// TwinCAT 3 PLC project FLC
// ProgramVersion: 3.1.4026.12
// CompilerDefines: ABG
// libraries:
//   Tc2_IoFunctions, * (Beckhoff Automation GmbH)
//   Tc2_ModbusSrv, * (Beckhoff Automation GmbH)
//   Tc2_Standard, * (Beckhoff Automation GmbH)
//   Tc2_System, * (Beckhoff Automation GmbH)
//   Tc2_Utilities, * (Beckhoff Automation GmbH)
//   Tc3_Module, * (Beckhoff Automation GmbH)
//   EAP_Controller,1.0,LUA
//   Modbus_SPC,1.0,LUA
// project tree:
//   Functions/Communications/ EtherCAT_MappingEAP.TcPOU, EtherCAT_MappingModbus.TcPOU, Mapping_Monitoring_Variables.TcPOU, Mapping_Monitoring_Variables_ABG.TcPOU, Remap_EtherCAT_Variables.TcPOU
//   Functions/EventRecoder/ HistorianFunctionBlock.TcPOU, UnixTimestamp.TcPOU
//   Functions/Filters/ BandPassFilter.TcPOU, BandPassFilterParameters.TcPOU, BandPassFilterStruct.TcDUT, HighPassFilter.TcDUT, HPF_FilterInit.TcPOU, HPF_Function.TcPOU, LowPassFilter.TcDUT, LPF_FilterInit.TcPOU, LPF_Function.TcPOU
//   Functions/ Mapping_ModbusReadRegisters.TcPOU, Mapping_ModbusWriteRegisters.TcPOU, ModReadScaling.TcPOU
//   GlobalVar/ Communications.TcGVL, GlobalVar.TcGVL, GVL.TcGVL
//   Programs/ EAPControl.TcPOU, Timer.TcPOU, ModbusControl_Comm.TcPOU, State_Machine.TcPOU
//   Structures/Communication/EtherCAT/EAP Based Controller/EtherCAT/Commands Per Service/ AdditionalService_Struct_EAP.TcDUT, CommonBlock_Struct_EAP.TcDUT, FreqRegulation_Struct_EAP.TcDUT, InertiaEmulation_Struct_EAP.TcDUT, ModalFreq_Struct_EAP.TcDUT, VoltageRegulation_Struct_EAP.TcDUT
//   Structures/Communication/EtherCAT/EAP Based Controller/EtherCAT/Commands Per Service/Bits Per Commands/ Bits_AdditionalService_EAP.TcDUT, Bits_CommonBlock_EAP.TcDUT, Bits_FreqRegulation_EAP.TcDUT, Bits_InertiaEmulation_EAP.TcDUT, Bits_ModalFreq_EAP.TcDUT, Bits_VoltageRegulation_EAP.TcDUT
//   Structures/Communication/EtherCAT/EAP Based Controller/EtherCAT/ Commands_EAP.TcDUT, Parameters_EAP.TcDUT
//   Structures/Communication/EtherCAT/EAP Based Controller/EtherCAT/Parameters Per Service/ AdditionalService_Param_Struct_EAP.TcDUT, CommonBlock_Param_Struct_EAP.TcDUT, FreqRegulation_Param_Struct_EAP.TcDUT, InertiaEmulation_Param_Struct_EAP.TcDUT, ModalFreq_Param_Struct_EAP.TcDUT, VoltageRegulation_Param_Struct_EAP.TcDUT
//   Structures/Communication/EtherCAT/ EtherCAT_Inputs.TcDUT, EtherCAT_Monitor_Variables.TcDUT, EtherCAT_Stat_Variables.TcDUT, PowerOfService_Struct.TcDUT
//   Structures/Communication/EtherCAT/Modbus Based Controller/EtherCAT/Commands Per Service/ AdditionalService_Struct.TcDUT, CommonBlock_Struct.TcDUT, FreqRegulation_Struct.TcDUT, InertiaEmulation_Struct.TcDUT, ModalFreq_Struct.TcDUT, VoltageRegulation_Struct.TcDUT
//   Structures/Communication/EtherCAT/Modbus Based Controller/EtherCAT/Commands Per Service/Bits Per Commands/ Bits_AdditionalService.TcDUT, Bits_CommonBlock.TcDUT, Bits_FreqRegulation.TcDUT, Bits_InertiaEmulation.TcDUT, Bits_ModalFreq.TcDUT, Bits_VoltageRegulation.TcDUT
//   Structures/Communication/EtherCAT/Modbus Based Controller/EtherCAT/ Commands.TcDUT, Parameters.TcDUT
//   Structures/Communication/EtherCAT/Modbus Based Controller/EtherCAT/Parameters Per Service/ AdditionalService_Param_Struct.TcDUT, CommonBlock_Param_Struct.TcDUT, FreqRegulation_Param_Struct.TcDUT, InertiaEmulation_Param_Struct.TcDUT, ModalFreq_Param_Struct.TcDUT, VoltageRegulation_Param_Struct.TcDUT
//   Structures/Communication/EtherCAT/Modbus Based Controller/ EtherCAT_INT_VALUES.TcDUT
//   Structures/Communication/EtherCAT/RemapForSLC/EAP_para/ AdditionalService_Param_Struct_EAP_DINT.TcDUT, CommonBlock_Param_Struct_EAP_DINT.TcDUT, FreqRegulation_Param_Struct_EAP_DINT.TcDUT, InertiaEmulation_Param_Struct_EAP_DINT.TcDUT, ModalFreq_Param_Struct_EAP_DINT.TcDUT, VoltageRegulation_Param_Struct_EAP_DINT.TcDUT
//   Structures/Communication/EtherCAT/RemapForSLC/ EtherCAT_Inputs_DINT.TcDUT, EtherCAT_Monitor_Variables_DINT.TcDUT, Parameters_DINT.TcDUT, Parameters_EAP_DINT.TcDUT
//   Structures/Communication/EtherCAT/RemapForSLC/Modbus_para/ AdditionalService_Param_Struct_DINT.TcDUT, CommonBlock_Param_Struct_DINT.TcDUT, FreqRegulation_Param_Struct_DINT.TcDUT, InertiaEmulation_Param_Struct_DINT.TcDUT, ModalFreq_Param_Struct_DINT.TcDUT, VoltageRegulation_Param_Struct_DINT.TcDUT
//   Structures/Communication/EtherCAT/Warning/ Warnings_FLC.TcDUT, Warning_FLC_DINT.TcDUT
//   Structures/Communication/Modbus/ ModbusHoldingRegs.TcDUT, ModbusRead.TcDUT, ModbusRead_NRG.TcDUT, ModbusWrite.TcDUT, ModbusWrite_NRG.TcDUT, ScaledModRead.TcDUT
//   Structures/EventRecorder/ EthercatDataPacket.TcDUT
//   Structures/EventRecorder/HistorianDataType/ DateTimetype.TcDUT
//   Structures/StateMachine/ eCurrentState.TcDUT, eFEC_CurrState.TcDUT, StateMachineCommand.TcDUT
//   Structures/Transformations/ abcSignal.TcDUT, alphabetaSignal.TcDUT, dqsignal.TcDUT
//   Tasks/ EAPControl_Task.TcTTO, ModbusComm.TcTTO, StateMachine.TcTTO, TimerTask.TcTTO
// real-time tasks:
//   TASK StateMachine: cycle T#5ms, priority 8, ADS port 350
//   TASK ModbusComm: cycle T#20ms, priority 12, ADS port 351
//   TASK TimerTask: cycle T#1ms, priority 6, ADS port 353
//   TASK EAPControl_Task: cycle T#800us, priority 4, ADS port 354
//   TASK PlcTask: cycle T#10ms, priority 10, ADS port 352
// I/O:
//   DEVICE Device 1 (EtherCAT Slave), AmsNetId 10.150.0.126.2.255
// variable links:
//   FLC/FLC Instance <-> Device 1 (EtherCAT Slave)
//     EAPControl_Task Inputs/Communications.EtherCAT_Commands <-> Inputs/Commands Modbus
//     ModbusComm Inputs/Communications.EtherCAT_EAP_Commands <-> Inputs/Commands EAP
//     StateMachine Inputs/Communications.EhterCAT_Parameters_DINT <-> Inputs/Modbus_parameters
//     StateMachine Inputs/Communications.EtherCAT_EAP_Parameters_DINT <-> Inputs/EAP_paramteres
//     StateMachine Inputs/Communications.EtherCAT_Inputs_DINT <-> Inputs/EtherCAT_inputs
//     StateMachine Outputs/Communications.EtherCAT_Monitor_Variables_DINT <-> Outputs/Mornitoring Information
//     StateMachine Outputs/Communications.EtherCAT_Variables <-> Outputs/Status
//     StateMachine Outputs/Communications.PowerOfService <-> Outputs/PowerOfservices
//     TimerTask Inputs/GVL.TransmitApproved <-> Inputs/EventRecorderApproved
//     TimerTask Outputs/GVL.HistorianDataPacket_EtherCAT <-> Outputs/EventRecorder

CONFIGURATION FLC
    RESOURCE PLC ON TwinCAT3
        TASK EAPControl_Task(INTERVAL := T#800us, PRIORITY := 4);
        TASK ModbusComm(INTERVAL := T#20ms, PRIORITY := 12);
        TASK StateMachine(INTERVAL := T#5ms, PRIORITY := 8);
        TASK TimerTask(INTERVAL := T#1ms, PRIORITY := 6);
        PROGRAM EAPControl WITH EAPControl_Task : EAPControl;
        PROGRAM ModbusControl_Comm WITH ModbusComm : ModbusControl_Comm;
        PROGRAM State_Machine WITH StateMachine : State_Machine;
        PROGRAM Timer WITH TimerTask : Timer;
    END_RESOURCE
END_CONFIGURATION

// ---- Functions/Filters/BandPassFilterStruct.TcDUT
TYPE BandPassFilterStruct :
STRUCT
	G1_a0 : REAL;
	G1_a1 : REAL;
	G1_a2 : REAL;

	G1_b0 : REAL;
	
	output : REAL;
	error1 : REAL;
	error2 : REAL;
	output1 : REAL;
	output2 : REAL;

END_STRUCT
END_TYPE

// ---- Functions/Filters/HighPassFilter.TcDUT
TYPE HighPassFilter :
STRUCT
	FrequencyCut: REAL;
	Den: REAL;
	CutFreq: REAL;
	a1: REAL;
	b0: REAL;
	b1: REAL;
	ErrorFilt: REAL;
	OutputFilt: REAL;
END_STRUCT
END_TYPE

// ---- Functions/Filters/LowPassFilter.TcDUT
TYPE LowPassFilter :
STRUCT
	FrequencyCut: REAL;
	Den: REAL;
	CutFreq: REAL;
	a1: REAL;
	b0: REAL;
	b1: REAL;
	ErrorFilt: REAL;
	OutputFilt: REAL;
END_STRUCT
END_TYPE

// ---- Structures/Communication/EtherCAT/EAP Based Controller/EtherCAT/Commands Per Service/AdditionalService_Struct_EAP.TcDUT
TYPE AdditionalService_Struct_EAP :
UNION
		Value : INT;
		Bits : Bits_CommonBlock;
END_UNION
END_TYPE

// ---- Structures/Communication/EtherCAT/EAP Based Controller/EtherCAT/Commands Per Service/Bits Per Commands/Bits_AdditionalService_EAP.TcDUT
TYPE Bits_AdditionalService_EAP :
STRUCT
	//Additional Service
		Reserved1 : 	BIT;	//0
		Reserved2 : 	BIT;	//1
		Reserved3 : 	BIT;	//2
		Reserved4 : 	BIT;	//3
		Reserved5 : 	BIT;	//4
		Reserved6 : 	BIT;	//5
		Reserved7 : 	BIT;	//6
		Reserved8 : 	BIT;	//7
		Reserved9 : 	BIT;	//8
		Reserved10 : 	BIT;	//9
		Reserved11 : 	BIT;	//10
		Reserved12 : 	BIT;	//11
		Reserved13 : 	BIT;	//12
		Reserved14 : 	BIT;	//13
		Reserved15 : 	BIT;	//14
		Reserved16 : 	BIT;	//15
END_STRUCT
END_TYPE

// ---- Structures/Communication/EtherCAT/EAP Based Controller/EtherCAT/Commands Per Service/Bits Per Commands/Bits_CommonBlock_EAP.TcDUT
TYPE Bits_CommonBlock_EAP :
STRUCT
	//Common Block
	ActivePowerLimitation : BIT;		//0
	ReactivePowerLimitation : BIT;		//1
	Delta_Limitation : BIT; 			//2
	E_Limitation : BIT; 				//3
	SOC_Limitation : BIT;				//4
	Reset_To_Default_Common : BIT;		//5
	Reserved1 : BIT;					//6
	Reserved2 : BIT;					//7
	Reserved3 : BIT;					//8
	Reserved4 : BIT;					//9
	Reserved5 : BIT;					//10
	Reserved6 : BIT;					//11
	Reserved7 : BIT;					//12
	Reserved8 : BIT;					//13
	Reserved9 : BIT;					//14
	Reserved10 : BIT;					//15
END_STRUCT
END_TYPE

// ---- Structures/Communication/EtherCAT/EAP Based Controller/EtherCAT/Commands Per Service/Bits Per Commands/Bits_FreqRegulation_EAP.TcDUT
TYPE Bits_FreqRegulation_EAP :
STRUCT
	//Frequency Regulation
		Enable_DroopP : BIT;						//0
		Enable_DeadBandFreq : BIT;					//1
		Delta_Power_Limitation_freq : BIT;			//2
		Delta_Energy_Limitation : BIT;				//3
		Reset_To_Default_Freq : BIT;				//4
		Reserved1 : BIT;							//5
		Reserved2 : BIT;							//6
		Reserved3 : BIT;							//7
		Reserved4 : BIT;							//8
		Reserved5 : BIT;							//9
		Reserved6 : BIT;							//10
		Reserved7 : BIT;							//11
		Reserved8 : BIT;							//12
		Reserved9 : BIT;							//13
		Reserved10 : BIT;							//14
		Reserved11 : BIT;							//15
END_STRUCT
END_TYPE

// ---- Structures/Communication/EtherCAT/EAP Based Controller/EtherCAT/Commands Per Service/Bits Per Commands/Bits_InertiaEmulation_EAP.TcDUT
TYPE Bits_InertiaEmulation_EAP :
STRUCT
	//Inertia Emulation
	Enable_Inertia : BIT;					//0
	Reset_States_Inertia : BIT;				//1
	ROCOF_Limitation : BIT;					//2
	Reset_To_Default_Inertia : BIT;			//3
	Reserved1 : BIT;						//4
	Reserved2 : BIT;						//5
	Reserved3 : BIT;						//6
	Reserved4 : BIT;						//7
	Reserved5 : BIT;						//8
	Reserved6 : BIT;						//9
	Reserved7 : BIT;						//10
	Reserved8 : BIT;						//11
	Reserved9 : BIT;						//12
	Reserved10 : BIT;						//13
	Reserved11 : BIT;						//14
	Reserved12 : BIT;						//15
END_STRUCT
END_TYPE

// ---- Structures/Communication/EtherCAT/EAP Based Controller/EtherCAT/Commands Per Service/Bits Per Commands/Bits_ModalFreq_EAP.TcDUT
TYPE Bits_ModalFreq_EAP :
STRUCT
	//Modal Frequency Attenuation
		Enable_ModalFreq : BIT;						//0
		ModalFreq_PowerLimitation : BIT;			//1
		ROCOF_Limitation_ModalFreq : BIT;			//2
		Reset_To_Default_ModalFreq : BIT;			//3
		Reserved1 : BIT;							//4
		Reserved2 : BIT;							//5
		Reserved3 : BIT;							//6
		Reserved4 : BIT;							//7
		Reserved5 : BIT;							//8
		Reserved6 : BIT;							//9
		Reserved7 : BIT;							//10
		Reserved8 : BIT;							//11
		Reserved9 : BIT;							//12
		Reserved10 : BIT;							//13
		Reserved11 : BIT;							//14
		Reserved12 : BIT;							//15
END_STRUCT
END_TYPE

// ---- Structures/Communication/EtherCAT/EAP Based Controller/EtherCAT/Commands Per Service/Bits Per Commands/Bits_VoltageRegulation_EAP.TcDUT
TYPE Bits_VoltageRegulation_EAP :
STRUCT
	//Voltage Regulation
		Enable_VoltageRegulation : BIT;					//0
		Delta_Power_Limitation_VoltReg : BIT;			//1
		Enable_deadBandV : BIT;					//2
		Reset_To_Default_VoltReg : BIT;			//3
		Reserved1 : BIT;							//4
		Reserved2 : BIT;							//5
		Reserved3 : BIT;							//6
		Reserved4 : BIT;							//7
		Reserved5 : BIT;							//8
		Reserved6 : BIT;							//9
		Reserved7 : BIT;							//10
		Reserved8 : BIT;							//11
		Reserved9 : BIT;							//12
		Reserved10 : BIT;							//13
		Reserved11 : BIT;							//14
		Reserved12 : BIT;							//15
END_STRUCT
END_TYPE

// ---- Structures/Communication/EtherCAT/EAP Based Controller/EtherCAT/Commands Per Service/CommonBlock_Struct_EAP.TcDUT
TYPE CommonBlock_Struct_EAP :
UNION
	Value : INT;
	Bits : Bits_CommonBlock_EAP;
END_UNION
END_TYPE

// ---- Structures/Communication/EtherCAT/EAP Based Controller/EtherCAT/Commands Per Service/FreqRegulation_Struct_EAP.TcDUT
TYPE FreqRegulation_Struct_EAP :
UNION
	Value : INT;
	Bits : Bits_FreqRegulation_EAP;
END_UNION
END_TYPE

// ---- Structures/Communication/EtherCAT/EAP Based Controller/EtherCAT/Commands Per Service/InertiaEmulation_Struct_EAP.TcDUT
TYPE InertiaEmulation_Struct_EAP :
UNION
		Value : INT;
		Bits : Bits_InertiaEmulation_EAP;
END_UNION
END_TYPE

// ---- Structures/Communication/EtherCAT/EAP Based Controller/EtherCAT/Commands Per Service/ModalFreq_Struct_EAP.TcDUT
TYPE ModalFreq_Struct_EAP :
UNION
		Value : INT;
		Bits : Bits_ModalFreq_EAP;
END_UNION
END_TYPE

// ---- Structures/Communication/EtherCAT/EAP Based Controller/EtherCAT/Commands Per Service/VoltageRegulation_Struct_EAP.TcDUT
TYPE VoltageRegulation_Struct_EAP :
UNION
	Value : INT;
	Bits : Bits_VoltageRegulation_EAP;
END_UNION
END_TYPE

// ---- Structures/Communication/EtherCAT/EAP Based Controller/EtherCAT/Commands_EAP.TcDUT
TYPE Commands_EAP :
STRUCT
	//Common Block
		CommonBlock_EAP : CommonBlock_Struct_EAP;
	//Inertia Commands
		InertiaEmulation_EAP : InertiaEmulation_Struct_EAP;
	//Frequecy Regulation
		FrequencyRegulation_EAP : FreqRegulation_Struct_EAP;
	//Modal Frequencies attenuation
		ModalFreq_EAP : ModalFreq_Struct_EAP;
	//Voltage Regulation
		VoltageRegulation_EAP : VoltageRegulation_Struct_EAP;
	//Additional Service
		AddtionalService_EAP : AdditionalService_Struct_EAP;
END_STRUCT
END_TYPE

// ---- Structures/Communication/EtherCAT/EAP Based Controller/EtherCAT/Parameters Per Service/AdditionalService_Param_Struct_EAP.TcDUT
TYPE AdditionalService_Param_Struct_EAP :
STRUCT
	//Additional Service
		Reserved1 : 	REAL;	//0
		Reserved2 : 	REAL;	//1
		Reserved3 : 	REAL;	//2
		Reserved4 : 	REAL;	//3
		Reserved5 : 	REAL;	//4
		Reserved6 : 	REAL;	//5
		Reserved7 : 	REAL;	//6
		Reserved8 : 	REAL;	//7
		Reserved9 : 	REAL;	//8
		Reserved10 : 	REAL;	//9
		Reserved11 : 	REAL;	//10
		Reserved12 : 	REAL;	//11
		Reserved13 : 	REAL;	//12
		Reserved14 : 	REAL;	//13
		Reserved15 : 	REAL;	//14
		Reserved16 : 	REAL;	//15
END_STRUCT
END_TYPE

// ---- Structures/Communication/EtherCAT/EAP Based Controller/EtherCAT/Parameters Per Service/CommonBlock_Param_Struct_EAP.TcDUT
TYPE CommonBlock_Param_Struct_EAP :
STRUCT
	//Common Block parameters
		NominalPower : REAL := 1E6;			//0
		NominalFreq : REAL := 400;			//1
		NominalVolt : REAL := 50;			//2
		ActivePowerLimit : REAL := 1E6;		//3
		ReactivePowerLimit: REAL := 1E6;	//4
		Delta_limits : REAL := 1;			//5
		E_Limits : REAL := 200;				//6
		Kp_ReactiveControl : REAL := 1E-4;	//7
		Ki_ReactiveControl : REAL := 1E-4;	//8
		VirtualReactance : REAL := 0.3;		//9
		VirtualResistor : REAL := 0.1;		//10
		Reserved1 : REAL;					//11
		Reserved2 : REAL;					//12
		Reserved3 : REAL;					//13
		Reserved4 : REAL;					//14
		Reserved5 : REAL;					//15
END_STRUCT
END_TYPE

// ---- Structures/Communication/EtherCAT/EAP Based Controller/EtherCAT/Parameters Per Service/FreqRegulation_Param_Struct_EAP.TcDUT
TYPE FreqRegulation_Param_Struct_EAP :
STRUCT
	//Frequency Regulation
		DroopConstantP : REAL := 4;			//0
		Max_Delta_Energy : REAL := 1E6;		//1
		PowerLimit_Freq : REAL := 1E6;			//2
		LowPassFilter_CutOff_Freq : REAL := 1;			//3
		DeadBand_Limits_P : REAL := 30;			//4
		Reserved1 : REAL;				//5
		Reserved2 : REAL;				//6	
		Reserved3 : REAL;				//7
		Reserved4 : REAL;				//8
		Reserved5 : REAL;				//9
		Reserved6 : REAL;				//10
		Reserved7 : REAL;				//11
		Reserved8 : REAL;				//12
		Reserved9 : REAL;				//13
		Reserved10 : REAL;				//14
		Reserved11 : REAL;				//15
END_STRUCT
END_TYPE

// ---- Structures/Communication/EtherCAT/EAP Based Controller/EtherCAT/Parameters Per Service/InertiaEmulation_Param_Struct_EAP.TcDUT
TYPE InertiaEmulation_Param_Struct_EAP :
STRUCT
	//Inertia Emulation
		Inertia_Constant : REAL := 5;		//0
		Damping_Constant : REAL := 0.7;		//1
		HighPassFilterConst : REAL := 0.1;		//2
		Max_ROCOF : REAL := 6;				//3
		Reserved1 : REAL;				//4
		Reserved2 : REAL;				//5	
		Reserved3 : REAL;				//6
		Reserved4 : REAL;				//7
		Reserved5 : REAL;				//8
		Reserved6 : REAL;				//9
		Reserved7 : REAL;				//10
		Reserved8 : REAL;				//11
		Reserved9 : REAL;				//12
		Reserved10 : REAL;				//13
		Reserved11 : REAL;				//14
		Reserved12 : REAL;				//15
END_STRUCT
END_TYPE

// ---- Structures/Communication/EtherCAT/EAP Based Controller/EtherCAT/Parameters Per Service/ModalFreq_Param_Struct_EAP.TcDUT
TYPE ModalFreq_Param_Struct_EAP :
STRUCT
	//Modal Frequency Attenuation
		ModalFreq_Gain : REAL := 1000;				//0
		ModalFreq_PowerLimit : REAL := 1E6;		//1
		Max_ROCOF_Modal : REAL := 6;				//2
		BandPassFilter_CenterFreq : REAL := 5;	//3
		Reserved1 : REAL;					//4
		Reserved2 : REAL;					//5	
		Reserved3 : REAL;					//6
		Reserved4 : REAL;					//7
		Reserved5 : REAL;					//8
		Reserved6 : REAL;					//9
		Reserved7 : REAL;					//10
		Reserved8 : REAL;					//11
		Reserved9 : REAL;					//12
		Reserved10 : REAL;					//13
		Reserved11 : REAL;					//14
		Reserved12 : REAL;					//15
END_STRUCT
END_TYPE

// ---- Structures/Communication/EtherCAT/EAP Based Controller/EtherCAT/Parameters Per Service/VoltageRegulation_Param_Struct_EAP.TcDUT
TYPE VoltageRegulation_Param_Struct_EAP :
STRUCT
	//Voltage Regulation
		DroopConstantQ : REAL := 20;			//0
		LowPassFilter_CutOff_Volt : REAL := 1;	//1
		DeadBand_Limit_Q : REAL := 20;			//2
		PowerLimit_Volt : REAL := 1E6;			//3
		Reserved1 : REAL;						//4
		Reserved2 : REAL;						//5
		Reserved3 : REAL;						//6
		Reserved4 : REAL;						//7
		Reserved5 : REAL;						//8
		Reserved6 : REAL;						//9
		Reserved7 : REAL;						//10
		Reserved8 : REAL;						//11
		Reserved9 : REAL;						//12
		Reserved10 : REAL;						//13
		Reserved11 : REAL;						//14
		Reserved12 : REAL;						//15
END_STRUCT
END_TYPE

// ---- Structures/Communication/EtherCAT/EAP Based Controller/EtherCAT/Parameters_EAP.TcDUT
TYPE Parameters_EAP :
STRUCT
	//Common Block
		CommonBlock_Params_EAP : CommonBlock_Param_Struct_EAP;
	//Inertia Emulation
		InertiaEmulation_Params_EAP : InertiaEmulation_Param_Struct_EAP;
	//Frequency Regulation
		FrequencyRegulation_Params_EAP : FreqRegulation_Param_Struct_EAP;
	//Modal Frequencies Attenunation
		ModalFrequency_Params_EAP : ModalFreq_Param_Struct_EAP;
	//Voltage Regulation
		VoltageRegulation_Params_EAP : VoltageRegulation_Param_Struct_EAP;
	//Additional Service
		AdditonalSerivce : AdditionalService_Param_Struct_EAP;
END_STRUCT
END_TYPE

// ---- Structures/Communication/EtherCAT/EtherCAT_Inputs.TcDUT
{define JEMA}
TYPE EtherCAT_Inputs :
STRUCT
	Command : StateMachineCommand;				//0
	ActivePowerReference : REAL;				//1
	ReactivePowerReference : REAL;				//2
	Heartbeat : REAL;							//3
	Reserved4 : REAL;							//4
	Reserved5 : REAL;							//5
	Reserved6 : REAL;							//6
	Reserved7 : REAL;							//7
	Reserved8 : REAL;							//8
	Reserved9 : REAL;							//9	
	Reserved10 : REAL;							//10
	Reserved11 : REAL;							//11
	Reserved12 : REAL;							//12
	Reserved13 : REAL;							//13
	Reserved14 : REAL;							//14
	Reserved15 : REAL;							//15
END_STRUCT
END_TYPE

// ---- Structures/Communication/EtherCAT/EtherCAT_Monitor_Variables.TcDUT
TYPE EtherCAT_Monitor_Variables :
STRUCT
	BatSoc 			: REAL;				//0 - 100
	BatSocUpLim 	: REAL;				//1 - 100
	BatSocLowLim 	: REAL;				//2
	MaxWAval 		: REAL;				//3
	MaxWCharVal 	: REAL;				//4
	MaxVArAval 		: REAL;				//5
	MinVArAval 		: REAL;				//6
	TotW 			: REAL;				//7
	TotVAr 			: REAL;				//8
	GridFre 		: REAL;				//9
	Vrmsa 			: REAL;				//10
	Vrmsb 			: REAL;				//11
	Vrmsc 			: REAL;				//12
	Irmsa 			: REAL;				//13
	Irmsb 			: REAL;				//14
	Irmsc 			: REAL;				//15
END_STRUCT
END_TYPE

// ---- Structures/Communication/EtherCAT/EtherCAT_Stat_Variables.TcDUT
TYPE EtherCAT_Stat_Variables :
STRUCT
	Status : DINT;				//0
	HeartBeat : DINT;			//1
	Alarms1 : DINT;				//2
	Alarms2 : DINT;				//3
	Alarms3 : DINT;				//4
	Alarms4 : DINT;				//5
	WarningLog : Warning_FLC_DINT;	//6
	Reserved2 : DINT;			//7
END_STRUCT
END_TYPE

// ---- Structures/Communication/EtherCAT/Modbus Based Controller/EtherCAT/Commands Per Service/AdditionalService_Struct.TcDUT
TYPE AdditionalService_Struct :
UNION
		Value : INT;
		Bits : Bits_CommonBlock;
END_UNION
END_TYPE

// ---- Structures/Communication/EtherCAT/Modbus Based Controller/EtherCAT/Commands Per Service/Bits Per Commands/Bits_AdditionalService.TcDUT
TYPE Bits_AdditionalService :
STRUCT
	//Additional Service
		Reserved1 : 	BIT;	//0
		Reserved2 : 	BIT;	//1
		Reserved3 : 	BIT;	//2
		Reserved4 : 	BIT;	//3
		Reserved5 : 	BIT;	//4
		Reserved6 : 	BIT;	//5
		Reserved7 : 	BIT;	//6
		Reserved8 : 	BIT;	//7
		Reserved9 : 	BIT;	//8
		Reserved10 : 	BIT;	//9
		Reserved11 : 	BIT;	//10
		Reserved12 : 	BIT;	//11
		Reserved13 : 	BIT;	//12
		Reserved14 : 	BIT;	//13
		Reserved15 : 	BIT;	//14
		Reserved16 : 	BIT;	//15
END_STRUCT
END_TYPE

// ---- Structures/Communication/EtherCAT/Modbus Based Controller/EtherCAT/Commands Per Service/Bits Per Commands/Bits_CommonBlock.TcDUT
TYPE Bits_CommonBlock :
STRUCT
	//Common Block
		ActivePowerLimitation : 	BIT; 		//0
		ReactivePowerLimitation : 	BIT; 		//1
		State_Of_Health : 			BIT := 1;		//2
		Reset_To_Default_Common : 	BIT;		//3
		Reserved1 : 				BIT;		//4
		Reserved2 : 				BIT;		//5
		Reserved3 : 				BIT;		//6
		Reserved4 : 				BIT;		//7
		Reserved5 : 				BIT;		//8
		Reserved6 : 				BIT;		//9
		Reserved7 : 				BIT;		//10
		Reserved8 : 				BIT;		//11
		Reserved9 : 				BIT;		//12
		Reserved10 :			 	BIT;		//13
		Reserved11 : 				BIT;		//14
		Reserved12 : 				BIT;		//15
END_STRUCT
END_TYPE

// ---- Structures/Communication/EtherCAT/Modbus Based Controller/EtherCAT/Commands Per Service/Bits Per Commands/Bits_FreqRegulation.TcDUT
TYPE Bits_FreqRegulation :
STRUCT
	//Frequency Regulation
		Enable_DroopP : 					BIT;	//0
		Delta_Power_Limit_FreqRegulation : 	BIT;	//1
		Delta_Energy_Limit : 				BIT;	//2
		Reset_Energy_State : 				BIT;	//3
		DeadBandLimitationP :				BIT;	//4
		Reset_To_Default_FreqRegulation : 	BIT; 	//5
		Reserved1 : 						BIT;	//6
		Reserved2 : 						BIT;	//7
		Reserved3 : 						BIT;	//8
		Reserved4 : 						BIT;	//9
		Reserved5 : 						BIT;	//10
		Reserved6 : 						BIT;	//11
		Reserved7 : 						BIT;	//12
		Reserved8 : 						BIT;	//13
		Reserved9 : 						BIT;	//14
		Reserved10 : 						BIT;	//15
END_STRUCT
END_TYPE

// ---- Structures/Communication/EtherCAT/Modbus Based Controller/EtherCAT/Commands Per Service/Bits Per Commands/Bits_InertiaEmulation.TcDUT
TYPE Bits_InertiaEmulation :
STRUCT
	//Inertia Emulation
		Enable_Inertia : 			BIT;		//0
		Inertia_Reset_States : 		BIT;		//1
		Limit_ROCOF : 				BIT;		//2
		Delta_Power_Limit_Inertia : BIT;		//3
		Reset_To_Default_Inertia : 	BIT;		//4
		Reserved1 : 				BIT;		//5
		Reserved2 : 				BIT;		//6
		Reserved3 : 				BIT;		//7
		Reserved4 : 				BIT;		//8
		Reserved5 : 				BIT;		//9
		Reserved6 : 				BIT;		//10
		Reserved7 : 				BIT;		//11
		Reserved8 : 				BIT;		//12
		Reserved9 : 				BIT;		//13
		Reserved10 : 				BIT;		//14
		Reserved11 : 				BIT;		//15
END_STRUCT
END_TYPE

// ---- Structures/Communication/EtherCAT/Modbus Based Controller/EtherCAT/Commands Per Service/Bits Per Commands/Bits_ModalFreq.TcDUT
TYPE Bits_ModalFreq :
STRUCT
	//Modal Frequency Attenuation
		Enable_ModalFreq : 				BIT;	//0
		Delta_Power_Limit_ModalFreq : 	BIT;	//1
		Reset_To_Default_ModalFreq : 	BIT;	//2
		Reserved1 : 					BIT;	//3
		Reserved2 : 					BIT;	//4
		Reserved3 : 					BIT;	//5
		Reserved4 : 					BIT;	//6
		Reserved5 : 					BIT;	//7
		Reserved6 : 					BIT;	//8
		Reserved7 : 					BIT;	//9
		Reserved8 : 					BIT;	//10
		Reserved9 : 					BIT;	//11
		Reserved10 : 					BIT;	//12
		Reserved11 : 					BIT;	//13
		Reserved12 : 					BIT;	//14
		Reserved13 : 					BIT;	//15
END_STRUCT
END_TYPE

// ---- Structures/Communication/EtherCAT/Modbus Based Controller/EtherCAT/Commands Per Service/Bits Per Commands/Bits_VoltageRegulation.TcDUT
TYPE Bits_VoltageRegulation :
STRUCT
	//Voltage Regulation
		Enable_VoltageRef : 			BIT;	//0
		Delta_Power_Limit_Voltage : 	BIT;	//1
		DeadBandLimitationV : 			BIT;	//2
		Reset_To_Default_VoltageReg : 	BIT;	//3
		Reserved1 : 					BIT;	//4
		Reserved2 : 					BIT;	//5
		Reserved3 : 					BIT;	//6
		Reserved4 : 					BIT;	//7
		Reserved5 : 					BIT;	//8
		Reserved6 : 					BIT;	//9
		Reserved7 : 					BIT;	//10
		Reserved8 : 					BIT;	//11
		Reserved9 : 					BIT;	//12
		Reserved10 : 					BIT;	//13
		Reserved11 : 					BIT;	//14
		Reserved12 : 					BIT;	//15
END_STRUCT
END_TYPE

// ---- Structures/Communication/EtherCAT/Modbus Based Controller/EtherCAT/Commands Per Service/CommonBlock_Struct.TcDUT
TYPE CommonBlock_Struct :
UNION
		Value : INT;
		Bits : Bits_CommonBlock;
END_UNION
END_TYPE

// ---- Structures/Communication/EtherCAT/Modbus Based Controller/EtherCAT/Commands Per Service/FreqRegulation_Struct.TcDUT
TYPE FreqRegulation_Struct :
UNION
		Value : INT;
		Bits : Bits_FreqRegulation;
END_UNION
END_TYPE

// ---- Structures/Communication/EtherCAT/Modbus Based Controller/EtherCAT/Commands Per Service/InertiaEmulation_Struct.TcDUT
TYPE InertiaEmulation_Struct :
UNION
		Value : INT;
		Bits : Bits_InertiaEmulation;
END_UNION
END_TYPE

// ---- Structures/Communication/EtherCAT/Modbus Based Controller/EtherCAT/Commands Per Service/ModalFreq_Struct.TcDUT
TYPE ModalFreq_Struct :
UNION
		Value : INT;
		Bits : Bits_ModalFreq;
END_UNION
END_TYPE

// ---- Structures/Communication/EtherCAT/Modbus Based Controller/EtherCAT/Commands Per Service/VoltageRegulation_Struct.TcDUT
TYPE VoltageRegulation_Struct :
UNION
		Value : INT;
		Bits : Bits_VoltageRegulation;
END_UNION
END_TYPE

// ---- Structures/Communication/EtherCAT/Modbus Based Controller/EtherCAT/Commands.TcDUT
TYPE Commands :
STRUCT
	//Common Block
		CommonBlock : CommonBlock_Struct;
	//Inertia Commands
		InertiaEmulation : InertiaEmulation_Struct;
	//Frequecy Regulation
		FrequencyRegulation : FreqRegulation_Struct;
	//Modal Frequencies attenuation
		ModalFreq : ModalFreq_Struct;
	//Voltage Regulation
		VoltageRegulation : VoltageRegulation_Struct;
	//Additional Service
		AdditionalService : AdditionalService_Struct;
END_STRUCT
END_TYPE

// ---- Structures/Communication/EtherCAT/Modbus Based Controller/EtherCAT/Parameters Per Service/AdditionalService_Param_Struct.TcDUT
TYPE AdditionalService_Param_Struct :
STRUCT
	//Additional Service
		Reserved1 : 	REAL;	//0
		Reserved2 : 	REAL;	//1
		Reserved3 : 	REAL;	//2
		Reserved4 : 	REAL;	//3
		Reserved5 : 	REAL;	//4
		Reserved6 : 	REAL;	//5
		Reserved7 : 	REAL;	//6
		Reserved8 : 	REAL;	//7
		Reserved9 : 	REAL;	//8
		Reserved10 : 	REAL;	//9
		Reserved11 : 	REAL;	//10
		Reserved12 : 	REAL;	//11
		Reserved13 : 	REAL;	//12
		Reserved14 : 	REAL;	//13
		Reserved15 : 	REAL;	//14
		Reserved16 : 	REAL;	//15
END_STRUCT
END_TYPE

// ---- Structures/Communication/EtherCAT/Modbus Based Controller/EtherCAT/Parameters Per Service/CommonBlock_Param_Struct.TcDUT
TYPE CommonBlock_Param_Struct :
STRUCT
	//Common Block parameters
		NominalPower : REAL := 1E6;			//0
		NominalVoltage : REAL := 240;		//1
		NominalFreq : REAL := 50;			//2
		ActivePowerLimit : REAL := 1E6;		//3
		ReactivePowerLimit: REAL := 1E6;	//4
		Reserved1 : REAL;					//5
		Reserved2 : REAL;					//6
		Reserved3 : REAL;					//7
		Reserved4 : REAL;					//8
		Reserved5 : REAL;					//9
		Reserved6 : REAL;					//10
		Reserved7 : REAL;					//11
		Reserved8 : REAL;					//12
		Reserved9 : REAL;					//13
		Reserved10 : REAL;					//14
		Reserved11 : REAL;					//15
END_STRUCT
END_TYPE

// ---- Structures/Communication/EtherCAT/Modbus Based Controller/EtherCAT/Parameters Per Service/FreqRegulation_Param_Struct.TcDUT
TYPE FreqRegulation_Param_Struct :
STRUCT
	//Frequency Regulation
		DroopConstantP : REAL := 4;			//0
		Max_delta_Energy : REAL := 1E6;		//1
		PowerLimit_Freq : REAL := 1E6;		//2
		FrequencyCutOff : REAL := 0.2;		//3
		FreqDeadBand : REAL := 30;			//4
		Reserved1 : REAL;					//5
		Reserved2 : REAL;					//6	
		Reserved3 : REAL;					//7
		Reserved4 : REAL;					//8
		Reserved5 : REAL;					//9
		Reserved6 : REAL;					//10
		Reserved7 : REAL;					//11
		Reserved8 : REAL;					//12
		Reserved9 : REAL;					//13
		Reserved10 : REAL;					//14
		Reserved11 : REAL;					//15
END_STRUCT
END_TYPE

// ---- Structures/Communication/EtherCAT/Modbus Based Controller/EtherCAT/Parameters Per Service/InertiaEmulation_Param_Struct.TcDUT
TYPE InertiaEmulation_Param_Struct :
STRUCT
	//Inertia Emulation
		Inertia_Constant : REAL := 5;		//0
		HighPassFilterConst : REAL := 0.1;	//1
		Max_ROCOF : REAL := 5;				//2
		PowerLimit_Inertia : REAL := 1E6;	//3
		Reserved1 : REAL;					//4
		Reserved2 : REAL;					//5	
		Reserved3 : REAL;					//6
		Reserved4 : REAL;					//7
		Reserved5 : REAL;					//8
		Reserved6 : REAL;					//9
		Reserved7 : REAL;					//10
		Reserved8 : REAL;					//11
		Reserved9 : REAL;					//12
		Reserved10 : REAL;					//13
		Reserved11 : REAL;					//14
		Reserved12 : REAL;					//15
END_STRUCT
END_TYPE

// ---- Structures/Communication/EtherCAT/Modbus Based Controller/EtherCAT/Parameters Per Service/ModalFreq_Param_Struct.TcDUT
TYPE ModalFreq_Param_Struct :
STRUCT
	//Modal Frequency Attenuation
		ModalFreq_Gain : REAL := 1000;				//0
		BandPassFilter_CenterFreq : REAL := 31.4;	//1
		PowerLimit_ModalFreq : REAL := 1E6;		//2
		Reserved1 : REAL;					//3
		Reserved2 : REAL;					//4	
		Reserved3 : REAL;					//5
		Reserved4 : REAL;					//6
		Reserved5 : REAL;					//7
		Reserved6 : REAL;					//8
		Reserved7 : REAL;					//9
		Reserved8 : REAL;					//10
		Reserved9 : REAL;					//11
		Reserved10 : REAL;					//12
		Reserved11 : REAL;					//13
		Reserved12 : REAL;					//14
		Reserved13 : REAL;					//15
END_STRUCT
END_TYPE

// ---- Structures/Communication/EtherCAT/Modbus Based Controller/EtherCAT/Parameters Per Service/VoltageRegulation_Param_Struct.TcDUT
TYPE VoltageRegulation_Param_Struct :
STRUCT
	//Voltage Regulation
		DroopConstantV : REAL := 20;				//0
		PowerLimit_Voltage : REAL := 1E6;			//1
		VoltageCutOff : REAL := 0.1;				//2
		VoltDeadBand : REAL := 20;				//3
		Reserved1 : REAL;					//4
		Reserved2 : REAL;					//5
		Reserved3 : REAL;					//6
		Reserved4 : REAL;					//7
		Reserved5 : REAL;					//8
		Reserved6 : REAL;					//9
		Reserved7 : REAL;					//10
		Reserved8 : REAL;					//11
		Reserved9 : REAL;					//12
		Reserved10 : REAL;					//13
		Reserved11 : REAL;					//14
		Reserved12 : REAL;					//15
END_STRUCT
END_TYPE

// ---- Structures/Communication/EtherCAT/Modbus Based Controller/EtherCAT/Parameters.TcDUT
TYPE Parameters :
STRUCT
	//Common Block
		CommonBlock_Params : CommonBlock_Param_Struct;
	//Inertia Emulation
		InertiaEmulation_Params : InertiaEmulation_Param_Struct;
	//Frequency Regulation
		FrequencyRegulation_Params : FreqRegulation_Param_Struct;
	//Modal Frequencies Attenunation
		ModalFrequency_Params : ModalFreq_Param_Struct;
	//Voltage Regulation
		VoltageRegulation_Params : VoltageRegulation_Param_Struct;
	//Additional Service
		AdditionalService_Params : AdditionalService_Param_Struct;
END_STRUCT
END_TYPE

// ---- Structures/Communication/EtherCAT/Modbus Based Controller/EtherCAT_INT_VALUES.TcDUT
TYPE EtherCAT_INT_VALUES :
STRUCT
	TotW : INT;								//0
	TotVAr : INT;							//1
	Var1 : INT;						//2
	Var2 : INT;							//3
	Var3 : INT;							//4
	Var4 : INT;							//5
	Var5 : INT;							//6
	Var6 : INT;								//7
	Var7 : INT;								//8
	Var8 : INT;								//9
	Var9 : INT;								//10
	Var10 : INT;								//11
	Var11 : INT;								//12
	Var12 : INT;								//13
	Var13 : INT;								//14
	Var14 : INT;								//15
END_STRUCT
END_TYPE

// ---- Structures/Communication/EtherCAT/PowerOfService_Struct.TcDUT
TYPE PowerOfService_Struct :
STRUCT
	InertiaEmulationP_Service : REAL;
	FrequencyRegulationP_Service : REAL;
	ModalFreqAttP_Service : REAL;
	VoltageRegulationQ_Service : REAL;
END_STRUCT
END_TYPE

// ---- Structures/Communication/EtherCAT/RemapForSLC/EAP_para/AdditionalService_Param_Struct_EAP_DINT.TcDUT
TYPE AdditionalService_Param_Struct_EAP_DINT :
STRUCT
	//Additional Service
		Reserved1 : 	DINT;	//0
		Reserved2 : 	DINT;	//1
		Reserved3 : 	DINT;	//2
		Reserved4 : 	DINT;	//3
		Reserved5 : 	DINT;	//4
		Reserved6 : 	DINT;	//5
		Reserved7 : 	DINT;	//6
		Reserved8 : 	DINT;	//7
		Reserved9 : 	DINT;	//8
		Reserved10 : 	DINT;	//9
		Reserved11 : 	DINT;	//10
		Reserved12 : 	DINT;	//11
		Reserved13 : 	DINT;	//12
		Reserved14 : 	DINT;	//13
		Reserved15 : 	DINT;	//14
		Reserved16 : 	DINT;	//15
END_STRUCT
END_TYPE

// ---- Structures/Communication/EtherCAT/RemapForSLC/EAP_para/CommonBlock_Param_Struct_EAP_DINT.TcDUT
TYPE CommonBlock_Param_Struct_EAP_DINT :
STRUCT
	//Common Block parameters
		NominalPower 		: DINT := 1000000;			//0
		NominalFreq 		: DINT := 5000;			//1
		NominalVolt 		: DINT := 400;			//2
		ActivePowerLimit 	: DINT := 1000000;		//3
		ReactivePowerLimit	: DINT := 100000;	//4
		Delta_limits 		: DINT := 1;			//5
		E_Limits 			: DINT := 200;				//6
		Kp_ReactiveControl 	: DINT := 1000;	//1E-4;	//7
		Ki_ReactiveControl 	: DINT := 1000;	//1E-4;	//8
		VirtualReactance 	: DINT := 300;	//0.3		//9
		VirtualResistor 	: DINT := 100;	//0.1;		//10
		Reserved1 			: DINT;					//11
		Reserved2 			: DINT;					//12
		Reserved3 			: DINT;					//13
		Reserved4 			: DINT;					//14
		Reserved5 			: DINT;					//15
END_STRUCT
END_TYPE

// ---- Structures/Communication/EtherCAT/RemapForSLC/EAP_para/FreqRegulation_Param_Struct_EAP_DINT.TcDUT
TYPE FreqRegulation_Param_Struct_EAP_DINT :
STRUCT
	//Frequency Regulation
		DroopConstantP 		: DINT := 4;			//0
		Max_Delta_Energy 	: DINT := 1000000;		//1
		PowerLimit_Freq 	: DINT := 1000000;			//2
		LowPassFilter_CutOff_Freq : DINT := 1;			//3
		DeadBand_Limits_P 	: DINT := 30;			//4
		Reserved1 			: DINT;				//5
		Reserved2 			: DINT;				//6	
		Reserved3 			: DINT;				//7
		Reserved4 			: DINT;				//8
		Reserved5 			: DINT;				//9
		Reserved6 			: DINT;				//10
		Reserved7 			: DINT;				//11
		Reserved8 			: DINT;				//12
		Reserved9 			: DINT;				//13
		Reserved10 			: DINT;				//14
		Reserved11 			: DINT;				//15
END_STRUCT
END_TYPE

// ---- Structures/Communication/EtherCAT/RemapForSLC/EAP_para/InertiaEmulation_Param_Struct_EAP_DINT.TcDUT
TYPE InertiaEmulation_Param_Struct_EAP_DINT :
STRUCT
	//Inertia Emulation
		Inertia_Constant : DINT := 5;		//0
		Damping_Constant : DINT := 700;		//1
		HighPassFilterConst : DINT := 100;		//2
		Max_ROCOF : DINT := 6;				//3
		Reserved1 : DINT;				//4
		Reserved2 : DINT;				//5	
		Reserved3 : DINT;				//6
		Reserved4 : DINT;				//7
		Reserved5 : DINT;				//8
		Reserved6 : DINT;				//9
		Reserved7 : DINT;				//10
		Reserved8 : DINT;				//11
		Reserved9 : DINT;				//12
		Reserved10 : DINT;				//13
		Reserved11 : DINT;				//14
		Reserved12 : DINT;				//15
END_STRUCT
END_TYPE

// ---- Structures/Communication/EtherCAT/RemapForSLC/EAP_para/ModalFreq_Param_Struct_EAP_DINT.TcDUT
TYPE ModalFreq_Param_Struct_EAP_DINT :
STRUCT
	//Modal Frequency Attenuation
		ModalFreq_Gain : DINT := 1000;				//0
		ModalFreq_PowerLimit : DINT := 1000000;		//1
		Max_ROCOF_Modal : DINT := 6;				//2
		BandPassFilter_CenterFreq : DINT := 5;	//3
		Reserved1 : DINT;					//4
		Reserved2 : DINT;					//5	
		Reserved3 : DINT;					//6
		Reserved4 : DINT;					//7
		Reserved5 : DINT;					//8
		Reserved6 : DINT;					//9
		Reserved7 : DINT;					//10
		Reserved8 : DINT;					//11
		Reserved9 : DINT;					//12
		Reserved10 : DINT;					//13
		Reserved11 : DINT;					//14
		Reserved12 : DINT;					//15
END_STRUCT
END_TYPE

// ---- Structures/Communication/EtherCAT/RemapForSLC/EAP_para/VoltageRegulation_Param_Struct_EAP_DINT.TcDUT
TYPE VoltageRegulation_Param_Struct_EAP_DINT :
STRUCT
	//Voltage Regulation
		DroopConstantQ : DINT := 20;			//0
		LowPassFilter_CutOff_Volt : DINT := 1;	//1
		DeadBand_Limit_Q : DINT := 20;			//2
		PowerLimit_Volt : DINT := 1000000;		//3
		Reserved1 : DINT;						//4
		Reserved2 : DINT;						//5
		Reserved3 : DINT;						//6
		Reserved4 : DINT;						//7
		Reserved5 : DINT;						//8
		Reserved6 : DINT;						//9
		Reserved7 : DINT;						//10
		Reserved8 : DINT;						//11
		Reserved9 : DINT;						//12
		Reserved10 : DINT;						//13
		Reserved11 : DINT;						//14
		Reserved12 : DINT;						//15
END_STRUCT
END_TYPE

// ---- Structures/Communication/EtherCAT/RemapForSLC/EtherCAT_Inputs_DINT.TcDUT
TYPE EtherCAT_Inputs_DINT :
STRUCT
	Command : StateMachineCommand;				//0
	ActivePowerReference : DINT;				//1
	ReactivePowerReference : DINT;				//2
	Heartbeat : DINT;							//3
	Reserved4 : DINT;							//4
	Reserved5 : DINT;							//5
	Reserved6 : DINT;							//6
	Reserved7 : DINT;							//7
	Reserved8 : DINT;							//8
	Reserved9 : DINT;							//9	
	Reserved10 : DINT;							//10
	Reserved11 : DINT;							//11
	Reserved12 : DINT;							//12
	Reserved13 : DINT;							//13
	Reserved14 : DINT;							//14
	Reserved15 : DINT;							//15
END_STRUCT
END_TYPE

// ---- Structures/Communication/EtherCAT/RemapForSLC/EtherCAT_Monitor_Variables_DINT.TcDUT
TYPE EtherCAT_Monitor_Variables_DINT :
STRUCT
	BatSoc 			: DINT;				//0 - 100
	BatSocUpLim 	: DINT;				//1 - 100
	BatSocLowLim 	: DINT;				//2
	MaxWAval 		: DINT;				//3
	MaxWCharVal 	: DINT;				//4
	MaxVArAval 		: DINT;				//5
	MinVArAval 		: DINT;				//6
	TotW 			: DINT;				//7
	TotVAr 			: DINT;				//8
	GridFre 		: DINT;				//9
	Vrmsa 			: DINT;				//10
	Vrmsb 			: DINT;				//11
	Vrmsc 			: DINT;				//12
	Irmsa 			: DINT;				//13
	Irmsb 			: DINT;				//14
	Irmsc 			: DINT;				//15
END_STRUCT
END_TYPE

// ---- Structures/Communication/EtherCAT/RemapForSLC/Modbus_para/AdditionalService_Param_Struct_DINT.TcDUT
TYPE AdditionalService_Param_Struct_DINT :
STRUCT
	//Additional Service
		Reserved1 : 	DINT;	//0
		Reserved2 : 	DINT;	//1
		Reserved3 : 	DINT;	//2
		Reserved4 : 	DINT;	//3
		Reserved5 : 	DINT;	//4
		Reserved6 : 	DINT;	//5
		Reserved7 : 	DINT;	//6
		Reserved8 : 	DINT;	//7
		Reserved9 : 	DINT;	//8
		Reserved10 : 	DINT;	//9
		Reserved11 : 	DINT;	//10
		Reserved12 : 	DINT;	//11
		Reserved13 : 	DINT;	//12
		Reserved14 : 	DINT;	//13
		Reserved15 : 	DINT;	//14
		Reserved16 : 	DINT;	//15
END_STRUCT
END_TYPE

// ---- Structures/Communication/EtherCAT/RemapForSLC/Modbus_para/CommonBlock_Param_Struct_DINT.TcDUT
TYPE CommonBlock_Param_Struct_DINT :
STRUCT
	//Common Block parameters
		NominalPower : DINT := 1000000;			//0
		NominalVoltage : DINT := 240;			//1
		NominalFreq : DINT := 50;				//2
		ActivePowerLimit : DINT := 1000000;		//3
		ReactivePowerLimit: DINT := 1000000;	//4
		Reserved1 : DINT;					//5
		Reserved2 : DINT;					//6
		Reserved3 : DINT;					//7
		Reserved4 : DINT;					//8
		Reserved5 : DINT;					//9
		Reserved6 : DINT;					//10
		Reserved7 : DINT;					//11
		Reserved8 : DINT;					//12
		Reserved9 : DINT;					//13
		Reserved10 : DINT;					//14
		Reserved11 : DINT;					//15
END_STRUCT
END_TYPE

// ---- Structures/Communication/EtherCAT/RemapForSLC/Modbus_para/FreqRegulation_Param_Struct_DINT.TcDUT
TYPE FreqRegulation_Param_Struct_DINT :
STRUCT
	//Frequency Regulation
		DroopConstantP : DINT := 4;			//0
		Max_delta_Energy : DINT := 1000000;		//1
		PowerLimit_Freq : DINT := 1000000;		//2
		FrequencyCutOff : DINT := 200;		//3
		FreqDeadBand : DINT := 30;			//4
		Reserved1 : DINT;					//5
		Reserved2 : DINT;					//6	
		Reserved3 : DINT;					//7
		Reserved4 : DINT;					//8
		Reserved5 : DINT;					//9
		Reserved6 : DINT;					//10
		Reserved7 : DINT;					//11
		Reserved8 : DINT;					//12
		Reserved9 : DINT;					//13
		Reserved10 : DINT;					//14
		Reserved11 : DINT;					//15
END_STRUCT
END_TYPE

// ---- Structures/Communication/EtherCAT/RemapForSLC/Modbus_para/InertiaEmulation_Param_Struct_DINT.TcDUT
TYPE InertiaEmulation_Param_Struct_DINT :
STRUCT
	//Inertia Emulation
		Inertia_Constant : DINT := 5;		//0
		HighPassFilterConst : DINT := 100;	//1
		Max_ROCOF : DINT := 5;				//2
		PowerLimit_Inertia : DINT := 1000000;	//3
		Reserved1 : DINT;					//4
		Reserved2 : DINT;					//5	
		Reserved3 : DINT;					//6
		Reserved4 : DINT;					//7
		Reserved5 : DINT;					//8
		Reserved6 : DINT;					//9
		Reserved7 : DINT;					//10
		Reserved8 : DINT;					//11
		Reserved9 : DINT;					//12
		Reserved10 : DINT;					//13
		Reserved11 : DINT;					//14
		Reserved12 : DINT;					//15
END_STRUCT
END_TYPE

// ---- Structures/Communication/EtherCAT/RemapForSLC/Modbus_para/ModalFreq_Param_Struct_DINT.TcDUT
TYPE ModalFreq_Param_Struct_DINT :
STRUCT
	//Modal Frequency Attenuation
		ModalFreq_Gain : DINT := 1000;				//0
		BandPassFilter_CenterFreq : DINT := 31400;	//1
		PowerLimit_ModalFreq : DINT := 1000000;		//2
		Reserved1 : DINT;					//3
		Reserved2 : DINT;					//4	
		Reserved3 : DINT;					//5
		Reserved4 : DINT;					//6
		Reserved5 : DINT;					//7
		Reserved6 : DINT;					//8
		Reserved7 : DINT;					//9
		Reserved8 : DINT;					//10
		Reserved9 : DINT;					//11
		Reserved10 : DINT;					//12
		Reserved11 : DINT;					//13
		Reserved12 : DINT;					//14
		Reserved13 : DINT;					//15
END_STRUCT
END_TYPE

// ---- Structures/Communication/EtherCAT/RemapForSLC/Modbus_para/VoltageRegulation_Param_Struct_DINT.TcDUT
TYPE VoltageRegulation_Param_Struct_DINT :
STRUCT
	//Voltage Regulation
		DroopConstantV : DINT := 20;				//0
		PowerLimit_Voltage : DINT := 1000000;			//1
		VoltageCutOff : DINT := 100;				//2
		VoltDeadBand : DINT := 20;				//3
		Reserved1 : DINT;					//4
		Reserved2 : DINT;					//5
		Reserved3 : DINT;					//6
		Reserved4 : DINT;					//7
		Reserved5 : DINT;					//8
		Reserved6 : DINT;					//9
		Reserved7 : DINT;					//10
		Reserved8 : DINT;					//11
		Reserved9 : DINT;					//12
		Reserved10 : DINT;					//13
		Reserved11 : DINT;					//14
		Reserved12 : DINT;					//15
END_STRUCT
END_TYPE

// ---- Structures/Communication/EtherCAT/RemapForSLC/Parameters_DINT.TcDUT
TYPE Parameters_DINT :
STRUCT
	//Common Block
		CommonBlock_Params : CommonBlock_Param_Struct_DINT;
	//Inertia Emulation
		InertiaEmulation_Params : InertiaEmulation_Param_Struct_DINT;
	//Frequency Regulation
		FrequencyRegulation_Params : FreqRegulation_Param_Struct_DINT;
	//Modal Frequencies Attenunation
		ModalFrequency_Params : ModalFreq_Param_Struct_DINT;
	//Voltage Regulation
		VoltageRegulation_Params : VoltageRegulation_Param_Struct_DINT;
	//Additional Service
		AdditionalService_Params : AdditionalService_Param_Struct_DINT;
END_STRUCT
END_TYPE

// ---- Structures/Communication/EtherCAT/RemapForSLC/Parameters_EAP_DINT.TcDUT
TYPE Parameters_EAP_DINT :
STRUCT
	//Common Block
		CommonBlock_Params_EAP : CommonBlock_Param_Struct_EAP_DINT;
	//Inertia Emulation
		InertiaEmulation_Params_EAP : InertiaEmulation_Param_Struct_EAP_DINT;
	//Frequency Regulation
		FrequencyRegulation_Params_EAP : FreqRegulation_Param_Struct_EAP_DINT;
	//Modal Frequencies Attenunation
		ModalFrequency_Params_EAP : ModalFreq_Param_Struct_EAP_DINT;
	//Voltage Regulation
		VoltageRegulation_Params_EAP : VoltageRegulation_Param_Struct_EAP_DINT;
	//Additional Service
		AdditonalSerivce : AdditionalService_Param_Struct_EAP_DINT;
END_STRUCT
END_TYPE

// ---- Structures/Communication/EtherCAT/Warning/Warnings_FLC.TcDUT
TYPE Warnings_FLC :
STRUCT
	ModbusComm_FLC_PCS 				:		BIT; //0
	OverVoltage						: 		BIT; //1
	UnderVoltage					:		BIT; //2
	OverCurrent						:		BIT; //3
	OverFrequency					: 		BIT; //4
	UnderFrequency					:		BIT; //5
	CommandTimeout					:		BIT; //6
	Inertia_Overrange				:		BIT; //7
	Frequency_Overrange				:		BIT; //8
	VoltReg_Overrange				:		BIT; //9
	ModFreq_Overrange				:		BIT; //10
	Battery_80Perc					:		BIT; //11
	Battery_20Perc					:		BIT; //12
	EtherCAT_Failure				: 		BIT; //13
	Reserved2						: 		BIT; //14
	Reserved3						: 		BIT; //15
	Reserved4						: 		BIT; //16
	Reserved5						: 		BIT; //17
	Reserved6						: 		BIT; //18
	Reserved7						: 		BIT; //19
	Reserved8						: 		BIT; //20
	Reserved9						: 		BIT; //21
	Reserved10						: 		BIT; //22
	Reserved11						: 		BIT; //23
	Reserved12						: 		BIT; //24
	Reserved13						: 		BIT; //25
	Reserved14						: 		BIT; //26
	Reserved15						: 		BIT; //27
	Reserved16						: 		BIT; //28
	Reserved17						: 		BIT; //29
	Reserved18						: 		BIT; //30
	Reserved19						: 		BIT; //31
END_STRUCT
END_TYPE

// ---- Structures/Communication/EtherCAT/Warning/Warning_FLC_DINT.TcDUT
TYPE Warning_FLC_DINT :
UNION
	Value : DINT;
	Bits  : Warnings_FLC;
END_UNION
END_TYPE

// ---- Structures/Communication/Modbus/ModbusHoldingRegs.TcDUT
TYPE ModbusHoldingRegs :
STRUCT
		HoldRegsW	AT	%MB8192		:		FromSLC_1;		
		HoldRegsR	AT	%MB8704		:		To_SecondLevelControl;
END_STRUCT
END_TYPE

// ---- Structures/Communication/Modbus/ModbusRead.TcDUT
TYPE ModbusRead :
STRUCT
{IF defined (JEMA)}
	Vrmsa			:INT;	// 1, V, scale 1/10
	Vrmsb			:INT;	// 2, V, scale 1/10
	Vrmsc			:INT;	// 3, V, scale 1/10
	Irmsa			:INT;	// 4, A, scale 1/10
	Irmsb			:INT;	// 5, A, scale 1/10
	Irmsc			:INT;	// 6, A, scale 1/10
	TotW			:INT;	// 7, W, scale 10
	TotVAr			:INT;	// 8, W, scale 10
	GridFre			:INT;	// 9, Hz, scale 1/100
	HeartBeat		:UINT;  // 10
	GrAlm0			:UINT;	// 11, 1 flag 1 alarm
	GrAlm1			:UINT;	// 12
	GrAlm2			:UINT;	// 13
	GrAlm3			:UINT;	// 14
	GrAlm4			:UINT;	// 15
	BatSoc			:INT;	// 16, %
	BatSocUpLimit	:INT;	// 17, %
	BatSocLowLimit	:INT;	// 18, %
	fbOpMode		:UINT;  // 19
	CurOpMode		:UINT;  // 20
	fbP				:INT;	// 21, kW, 10
	fbQ				:INT;	// 22, kVar, 10		
	CtrlPriority 	:UINT; 	// 23, priority
	(* For connection with PLC*)
{ELSE}	
	fCommCommand		:REAL;
	BatSoc			 	:REAL;
	BatSocUpLim			:REAL;
	BatSocLowLim		:REAL;
	MaxWAval 			:REAL;
	MaxWCharval 		:REAL;
	MaxVArAval 			:REAL;
	MinVArAval			:REAL;
	TotW				:REAL;		// W
	TotVAr				:REAL;		// Var
	GridFre				:REAL;
	Vrmsa				:REAL;
	Vrmsb				:REAL;
	Vrmsc				:REAL;
	Irmsa				:REAL;
	Irmsb				:REAL;
	Irmsc				:REAL;
	//	Vsrfd				:REAL;
	//	Vsrfq				:REAL;
	HeartBeat			:UINT;
	DerOpMode			:UINT;
	GrAlm				:UDINT;
	AutoManCtl			:UINT;
	LocRemCtl			:UINT;
	OpModTest			:UINT;
	AutoManCtlFdbk		:UINT;
	LocRemCtlFdbk		:UINT;
	CtlSynVal			:UINT;
	RawP				:REAL;
	RawQ				:REAL;
	SM_ManualControl	:INT;		// 0 - FLC enabled  
{END_IF}	
END_STRUCT
END_TYPE

// ---- Structures/Communication/Modbus/ModbusRead_NRG.TcDUT
TYPE ModbusRead_NRG :
STRUCT
	TotW			:REAL;	// 7, W, scale 10
	TotVAr			:REAL;	// 8, W, scale 10
	
	Vrmsa			:REAL;	// 1, V, scale 1/10
	Vrmsb			:REAL;	// 2, V, scale 1/10
	Vrmsc			:REAL;	// 3, V, scale 1/10
	
	Irmsa			:INT;	// 4, A, scale 1/10
	Irmsb			:INT;	// 5, A, scale 1/10
	Irmsc			:INT;	// 6, A, scale 1/10
	
	fbOpMode		:INT;
	SignofCosineofPhi : INT;
	OutputApparentPower : INT;
	GridFre			:REAL;	// 9, Hz, scale 1/100
	
	BatSoc : INT;
	RawP				:REAL;	// 21, kW, 10
	RawQ				:REAL;	// 22, kVar, 10	
	HeartBeat		:UINT;  // 10
	fbOpMode2		:UINT;  // 19
	
	BatSocUpLimit	:INT;	// 17, %
	BatSocLowLimit	:INT;	// 18, %
	
	GrAlm1			:DINT;	// 12
	GrAlm2			:DINT;	// 13
	GrAlm3			:DINT;	// 14
	GrAlm0			:DINT;	// 15
	
END_STRUCT
END_TYPE

// ---- Structures/Communication/Modbus/ModbusWrite.TcDUT
TYPE ModbusWrite :
STRUCT
	{IF defined (JEMA)}
		Pset		:INT;	// 430, kW, scale 1
		Qset		:INT;	// 431, kVar, scale 1
		CmdOpMode	:INT;	// 432
		CurOpMode	:INT;	// 433
		HeartBeat	:UINT;	// 434
		R0			:INT;	// 435
		R1			:INT;	// 436
		R2			:INT;	// 437
		R3			:INT;	// 438
		(* For connection with PLC*)
	{ELSE}	
		wDerOpMode			:UINT;
		wAutoManCtl		 	:UINT;
		wLocRemCtl			:UINT;
		wOpModTest 			:UINT;
		CtlSynValfb			:UINT;
		HeartBeat			:UINT;
		OutWSet				:REAL;
		OutVArSet			:REAL;
		SLC_Debugger		:UINT;
		Reserved2			:REAL;
		Reserved3			:REAL;
		Reserved4			:REAL;
		(* For connection with DSP*)
	{END_IF}



	
END_STRUCT
END_TYPE

// ---- Structures/Communication/Modbus/ModbusWrite_NRG.TcDUT
TYPE ModbusWrite_NRG :
STRUCT
	CmdOpMode	:INT;	// 432
	Pset		:REAL;	// 430, kW, scale 1
	Qset		:REAL;	// 431, kVar, scale 1

END_STRUCT
END_TYPE

// ---- Structures/Communication/Modbus/ScaledModRead.TcDUT
TYPE ScaledModRead :
STRUCT
	Vrmsa			:REAL;	// 1, V, scale 1/10
	Vrmsb			:REAL;	// 2, V, scale 1/10
	Vrmsc			:REAL;	// 3, V, scale 1/10
	Irmsa			:REAL;	// 4, A, scale 1/10
	Irmsb			:REAL;	// 5, A, scale 1/10
	Irmsc			:REAL;	// 6, A, scale 1/10
	TotW			:REAL;	// 7, W, scale 10
	TotVAr			:REAL;	// 8, W, scale 10
	GridFre			:REAL;	// 9, Hz, scale 1/100
	HeartBeat		:UINT;  // 10
	GrAlm0			:UINT;	// 11, 1 flag 1 alarm
	
	GrAlm1			:UINT;	// 12
	GrAlm2			:UINT;	// 13
	GrAlm3			:UINT;	// 14
	GrAlm4			:UINT;	// 15
	BatSoc			:INT;	// 16, %
	BatSocUpLimit	:INT;	// 17, %
	BatSocLowLimit	:INT;	// 18, %
	fbOpMode		:UINT;  // 19
	CurOpMode		:UINT;  // 20
	fbP				:INT;	// 21, kW, 10
	fbQ				:INT;	// 22, kVar, 10		
	CtrlPriority 	:UINT; 	// 23, priority
	

//	Vd				:REAL;	// 22
//	Vq				:REAL;	// 23

//	Vdc				:REAL;   // 0, V, scale 1/10
//	Idc				:REAL;   // 0, V, scale 1/10		
END_STRUCT
END_TYPE

// ---- Structures/EventRecorder/EthercatDataPacket.TcDUT
TYPE EthercatDataPacket :
STRUCT
	TransmitRequest	:	INT;
	Index_TimeStamp	:	Index_TimeStamp;
	SingalIn_Modbus	:	EventRecorder_In_Modbus;
	SignalIn_EAP	:	EventRecorder_In_EAP;
	ControllerOut	:	EventRecorder_Controller_Output;
END_STRUCT
END_TYPE

// ---- Structures/EventRecorder/HistorianDataType/DateTimetype.TcDUT
TYPE DateTimetype :
UNION
	dwSecond	:	DWORD;
	dtSecond	:	DATE_AND_TIME;
END_UNION
END_TYPE

// ---- Structures/StateMachine/eCurrentState.TcDUT
{attribute 'qualified_only'}
//{attribute 'strict'}
TYPE eCurrentState :
(
	OFF := 0,
	STANDBY := 1,
	MANUAL := 2,
	AVG_PWR_CTR := 3,
	INST_PWR_CTR := 4
) INT;
END_TYPE

// ---- Structures/StateMachine/eFEC_CurrState.TcDUT
{attribute 'qualified_only'}
//{attribute 'strict'}
TYPE eFEC_CurrState :
(
	FEC_OFF := 1,
	FEC_PCS_START := 2,
	FEC_PCS_STOP := 3,
	FEC_STANDBY := 4,
	FEC_MANUAL := 5,
	FEC_AVG_PWR_CTR := 6,
	FEC_PCS_LOCAL_CONTROL := 7,
	FEC_RESERVED := 8,
	FEC_PCS_RAMPDOWN := 9,
	FEC_ALARM_STATE := 10,
	FEC_STANDBY_NoSwitching := 11,
	FEC_INST_PWR_CTR := 20
) INT;
END_TYPE

// ---- Structures/StateMachine/StateMachineCommand.TcDUT
{attribute 'qualified_only'}
//{attribute 'strict'}
TYPE StateMachineCommand :
(
	FEC_OFF := 0,
	FEC_STANDBY := 1,
	FEC_MANUAL := 2,
	FEC_AVG_PWR_CTR := 3
//	FEC_INST_PWR_CTR := 4
) DINT;
END_TYPE

// ---- Structures/Transformations/abcSignal.TcDUT
TYPE abcSignal :
STRUCT
	a	:	REAL;
	b	:	REAL;
	c	:	REAL;
END_STRUCT
END_TYPE

// ---- Structures/Transformations/alphabetaSignal.TcDUT
TYPE alphabetaSignal :
STRUCT
	alpha	:	REAL;
	beta	:	real;
END_STRUCT
END_TYPE

// ---- Structures/Transformations/dqsignal.TcDUT
TYPE dqsignal :
STRUCT
	d	:	REAL;
	q	:	REAL;
END_STRUCT
END_TYPE

// ---- GlobalVar/Communications.TcGVL
{attribute 'qualified_only'}
VAR_GLOBAL
	//Inputs
		//Modbus-Based Controller
			EtherCAT_Commands AT %I*: Commands;
			EhterCAT_Parameters	: Parameters;
			EhterCAT_Parameters_DINT AT %I*: Parameters_DINT;
		//EAP-Based Controller
			EtherCAT_EAP_Commands AT %I* : Commands_EAP;
			EtherCAT_EAP_Parameters  : Parameters_EAP;
			EtherCAT_EAP_Parameters_DINT AT %I* : Parameters_EAP_DINT;
		//EtherCAT Inputs	
			EtherCAT_Inputs : EtherCAT_Inputs;
			EtherCAT_Inputs_DINT AT %I*: EtherCAT_Inputs_DINT;	
		//EtherCAT Status Variables
			EtherCAT_Variables AT %Q* : EtherCAT_Stat_Variables;
		//EtherCAT Monitoring Variables
			EtherCAT_Monitor_Variables : EtherCAT_Monitor_Variables;
			EtherCAT_Monitor_Variables_DINT AT %Q* : EtherCAT_Monitor_Variables_DINT;
			
		//Service Outputs
			PowerOfService AT %Q* : PowerOfService_Struct;
			
		//EAP Recieve and Send Data
			EAP_Read AT %I* : data_16Real;
			EAP_Write AT %Q* : data_16Real;
			
		//Modbus Communication
			ModWriteNRG 		: 	ModbusWrite_NRG;
			ModReadNRG			: 	ModbusRead_NRG;
END_VAR

// ---- GlobalVar/GlobalVar.TcGVL
{attribute 'qualified_only'}
VAR_GLOBAL
	ModWrite 		: 	ModbusWrite;
	ModRead 		: 	ModbusRead;
	ScaledModRead	:	ScaledModRead;
	Vabcrms			:	abcSignal;
	Iabcrms			:	abcSignal;
	Pmodmeas		:	REAL;
	Qmodmeas		:	REAL;
	Pmodref			:	REAL;
	Qmodref			:	REAL;
	fgmeas			:	REAL;
	ModbusSPC_Enable: BOOL;
	EAP_SPC_Enable : BOOL;
	commandfromSLC	: (
		
			OFF := 0,
			STANDBY := 1,
			MANUAL := 2,
			AVG_PWR_CTR := 3,
			INST_PWR_CTR := 4);
	PreffromSLC	:	REAL;
	QreffromSLC	:	REAL;
	CommunicationFailureEtherCAT : BOOL;
	CommunicationFailureModbus : BOOL;
	MB_HoldingRegs	:	ModbusHoldingRegs;
	
	wMiliseconds : INT;
	HeartBeatFault : UINT;
	
	unixTime: UnixTimestamp;
    timestampSeconds: DateTimeType;
    timestampMilliseconds: UINT;
END_VAR

// ---- GlobalVar/GVL.TcGVL
{attribute 'qualified_only'}
VAR_GLOBAL
		// Event recorder
		fbHistorian	:	HistorianFunctionBlock;

		HistorianDataPacket_EtherCAT	AT	%Q* 	: EthercatDataPacket;
		TransmitApproved				AT	%I*		:	INT;
END_VAR

// ---- Programs/EAPControl.TcPOU
PROGRAM EAPControl
VAR
		SLCHeartBeat : REAL;
		CounterCommFailure : DINT;
		PRUEBAINT AT %I* : data_16bool;
		SPC_EAP : EAP_SPC;
		
		// Event recorder
		f	: 	REAL;
	t	:	REAL;
	va	:	REAL;
	vb	:	REAL;
	vc	:	REAL;
	EventRecorder_In_EAP	:	EventRecorder_In_EAP;
	RecordingTriger : BOOL	:= FALSE;
	
	EventRecorderControlOut	:	EventRecorder_Controller_Output;
	
	ER_HPF_power : HighPassFilter;
	Filtered_Power	:	REAL;
	
	ER_HPF_ReactivePower : HighPassFilter;
	Filtered_ReactivePower	:	REAL;
	
	
END_VAR

//Mapping EAP-Based Controller
	//IF GlobalVar.EAP_SPC_Enable THEN
		//EtherCAT_MappingEAP(ADR(SPC_EAP));
	//END_IF
	//IF GlobalVar.EAP_SPC_Enable = TRUE THEN
		SPC_EAP(ReferenceActivePower := Communications.EtherCAT_Inputs.ActivePowerReference,
				ReferenceReactivePower := Communications.EtherCAT_Inputs.ReactivePowerReference,
				ActivePowerMeasure := Communications.EAP_Read.var4,
				ReactivePowerMeasure := Communications.EAP_Read.var5,
				Va_inst := Communications.EAP_Read.var1,
				Vb_inst := Communications.EAP_Read.var2,
				Vc_inst := Communications.EAP_Read.var3,
				EnableControl := GlobalVar.EAP_SPC_Enable);
				
		Communications.EAP_Write.var1 := SPC_EAP.Global.SynchActivePower;
		Communications.EAP_Write.var2 := SPC_EAP.Global.SynchActivePower;
		Communications.EAP_Write.var3 := SPC_EAP.Global.SynchReactivePower;

	// Event Recorder trigger
		HPF_FilterInit(0.3, ADR(ER_HPF_Power), 800E-6);
		Filtered_Power := HPF_Function(Communications.EtherCAT_Monitor_Variables.TotW, ADR(ER_HPF_Power));
		
		HPF_FilterInit(0.3, ADR(ER_HPF_ReactivePower), 800E-6);
		Filtered_ReactivePower := HPF_Function(Communications.EtherCAT_Monitor_Variables.TotVAr, ADR(ER_HPF_ReactivePower));
		
		
		IF ABS(Filtered_power) > 50E3 OR ABS(Filtered_ReactivePower) > 50E3 OR Communications.EtherCAT_Commands.AdditionalService.Bits.Reserved1 THEN
			RecordingTriger := 1;
		ELSE
			RecordingTriger := 0;
		END_IF
		
	// Event Recorder
	gvl.fbHistorian.SetTtriger := RecordingTriger;
	
		f := 50;		// Hz
		t := t + 800E-6;
		
		va := LREAL_TO_REAL(SIN(2*PI*f*t));
		vb := LREAL_TO_REAL(SIN(2*PI*f*t - 2*PI/3));
		vc := LREAL_TO_REAL(SIN(2*PI*f*t + 2*PI/3));
		
		EventRecorder_In_EAP.Va := va;
		EventRecorder_In_EAP.Vb := vb;
		EventRecorder_In_EAP.Vc := vc;
		
		gvl.fbHistorian.ListeningRecording_IN_EAP(HistorianDataPacket := EventRecorder_In_EAP);
		
		
		
		IF Communications.EtherCAT_Inputs.Command = 4 THEN
			
			EventRecorderControlOut.Pref := 0.5*va;
			EventRecorderControlOut.Qref := 0.5*vc;
//			gvl.fbHistorian.ListeningRecording_ControlOut(HistorianDataPacket := EventRecorderControlOut);
		END_IF

END_PROGRAM

// ---- Functions/Filters/HPF_FilterInit.TcPOU
FUNCTION HPF_FilterInit : REAL
VAR_INPUT
	CutFreq : REAL;
	Filter : POINTER TO HighPassFilter;
	TS : REAL;
END_VAR
VAR
END_VAR

	Filter^.FrequencyCut := CutFreq;
	Filter^.CutFreq := 1/1/(2*3.1415*Filter^.FrequencyCut);
	
	Filter^.Den := 1/(TS + 2*(Filter^.CutFreq));	
	
	
	Filter^.a1 := (TS-2*Filter^.CutFreq)*Filter^.Den;
	Filter^.b0 := (2*Filter^.CutFreq)*Filter^.Den;
	Filter^.b1 := -(2*Filter^.CutFreq)*Filter^.Den;

END_FUNCTION

// ---- Functions/Filters/HPF_Function.TcPOU
FUNCTION HPF_Function : REAL
VAR_INPUT
	SignalToFilter : REAL;
	FilterParams : POINTER TO HighPassFilter;
END_VAR
VAR
END_VAR

HPF_Function := FilterParams^.b0*SignalToFilter + FilterParams^.b1*FilterParams^.ErrorFilt - FilterParams^.a1*Filterparams^.OutputFilt;

FilterParams^.ErrorFilt := SignalToFilter;
FilterParams^.OutputFilt := HPF_Function;

END_FUNCTION

// ---- Programs/ModbusControl_Comm.TcPOU
PROGRAM ModbusControl_Comm
VAR

//IP Adress
	ipAddr    		: STRING(15) := '10.200.8.195';		// Beckhoff FEC
	//ipAddr    		: STRING(15) := '10.200.8.217';		// Modicon PLC
	//ipAddr    		: STRING(15) := '192.168.1.51';		// JEMA DSP
	//ipAddr    		: STRING(15) := '169.254.227.11';	// NRG Board UPC
 	//ipAddr    		: STRING(15) := '10.200.8.196';		// NRG Board LUA
	//ipAddr    		: STRING(15) := '172.20.236.8';			// ABG
	
//Sampling time determination
	Tmod : INT;
	Tp : INT;
	Ts: REAL;
//Debug variables for modbus communication
 	DebugVar1  		: INT;			// Just for debugging
//Read and Write register for the modbus
 	fbWriteRegs 	: FB_MBWriteRegs;
	fbReadRegs		: FB_MBReadRegs;
 	bWriteRegs		: BOOL;
 	bReadRegs		: BOOL;
	pre_counter		:	DINT;
	SwapRW			: 	BOOL;
	mWritecounter:	DINT;
	mbreadcounter : UDINT := 1;
//Modbus-Based Controller system
	SPCModbus1 : modbus_SPC;
	ModbusSPC_Enable : BOOL;
//Voltage Calculation
	Vrmsmean: REAL;
//HeartBeat FEC and failure handling
	FECHeartBeat : DINT;
	CounterCommFailure : DINT;
	PreviousHeartBeat : UINT := 0;
	CounterFaultHeartBeat : UDINT;
	nQuantity: INT;
	
	
// Event recorder
	EventRecorder_in_modbus		:	EventRecorder_In_Modbus;
	EventRecorderControlOut		:	EventRecorder_Controller_Output;
	eventcnt	:	INT;
	
	Hugo :REAL;
	Hugo1 : INT;
	Hugo2 : INT;
	Hugo3: INT;
	Hugo4: INT;
	Hugo5 : INT;
	Hugo6 : INT;
	Hugo7 : INT;
	Hugo8 : INT;
END_VAR

//To write and read variables
//SwapRW := NOT SwapRW;
SwapRW := pre_counter = GlobalVar.ModRead.HeartBeat;

//Read Modbus Slave
	IF SwapRW AND (NOT fbReadRegs.bBusy) (*AND (NOT fbWriteRegs.bBusy) *) THEN
		mbreadcounter := 0;
		DebugVar1:= DebugVar1 + 1;			// Debuging variable
		
		{IF defined (JEMA)}
			Hugo1 := 1;
			ipAddr  := '192.168.1.51';
		{ELSE}
			Hugo1 := 2;		
			ipAddr  := '10.200.8.195';
		{END_IF}
		
		fbReadRegs.sIPAddr := ipAddr;
		
		fbReadRegs.nQuantity :=  SIZEOF(GlobalVar.ModRead)/2;
		
		{IF defined (JEMA)}
			Hugo2 := 1;
			fbReadRegs.nMBAddr :=  16#191;(*JEMA*)
			//fbReadRegs.nMBAddr :=(*16#0100;*)(*NRGLab*)
			//fbReadRegs.nMBAddr := 16#8000;//ABENGOA Memory location read
		{ELSE}
			Hugo2 := 2;	
			fbReadRegs.nMBAddr := 16#4100; //LUA-FEC 
		{END_IF}
			
		fbReadRegs.cbLength := SIZEOF(GlobalVar.ModRead);
		fbReadRegs.pDestAddr := ADR(GlobalVar.ModRead);
		fbReadRegs.tTimeout := T#5S;
		fbReadRegs(bExecute:=TRUE); 
	ELSE 
		fbReadRegs(bExecute:=FALSE);
		IF fbReadRegs.bBusy THEN
		mbreadcounter := mbreadcounter + 1;
		END_IF
	END_IF
//End of Read Modbus Slave

//Write Modbus Slave
	IF (NOT SwapRW) AND (NOT fbWriteRegs.bBusy) (*AND (NOT fbWriteRegs.bBusy)*) THEN
		//Scaling for Modbus Read
		
		{IF defined (JEMA)}
			Hugo3 := 1;
			ModreadScaling();
		{ELSE}	
			Hugo3 := 2;
		{END_IF}
		//Counter for synch
			pre_counter := GlobalVar.ModRead.HeartBeat;
		//RMS voltage calculation
			Vrmsmean := (GlobalVar.ModRead.Vrmsa + GlobalVar.ModRead.Vrmsb + GlobalVar.ModRead.Vrmsc)/3.0;
		//Heart Beat Failure
			IF GlobalVar.ModRead.HeartBeat = PreviousHeartBeat THEN
				CounterFaultHeartBeat := CounterFaultHeartBeat + 1;
			ELSE
				CounterFaultHeartBeat := 0;
			END_IF
			
			IF CounterFaultHeartBeat >= 5 THEN
				GlobalVar.HeartBeatFault := 1;
			ELSE
				GlobalVar.HeartBeatFault := 0;
			END_IF	
		//Sampling Time Calculation	
			Tmod := GlobalVar.wMiliseconds - Tp;
			IF Tmod<0 THEN Tmod:= (GlobalVar.wMiliseconds+1000)-Tp;
			Ts := Tmod*0.001;
			END_IF
			
		//IF GlobalVar.ModbusSPC_Enable THEN
			EtherCAT_MappingModbus(ADR(SPCModbus1));
		//END_IF
		
		//Enable Modbus-Based Controller
			IF GlobalVar.ModbusSPC_Enable = TRUE THEN
					SPCModbus1( 
					Pmodref := Communications.EtherCAT_Inputs.ActivePowerReference, 
					Qmodref := Communications.EtherCAT_Inputs.ReactivePowerReference,
					GridFre := Communications.EtherCAT_Monitor_Variables.GridFre*0.1591549430918,//CHECK BEFORE CONNECTION.
					Pmeasured := Communications.EtherCAT_Monitor_Variables.TotW,
					Qmeasured := Communications.EtherCAT_Monitor_Variables.TotVAr,
					Vmeasured := Communications.EtherCAT_Monitor_Variables.Vrmsa,
					//Control Parameters
					Ts := Ts,
					RampUpValue := 10,
					InertiaEmulationP=>Communications.PowerOfService.InertiaEmulationP_Service,
					FrequencyRegulationP => Communications.PowerOfService.FrequencyRegulationP_Service,
					ModalFreqAttP => Communications.PowerOfService.ModalFreqAttP_Service,		
					VoltageRegulationQ => Communications.PowerOfService.VoltageRegulationQ_Service,
					TestInertia := 1 //1 - Test mode ; 0- Normal Mode
					);
			//Output References from the controller
			{IF defined (JEMA)}
				Hugo4 := 1;
				GlobalVar.ModWrite.Pset := REAL_TO_INT(SPCModbus1.OutputP*0.001); //JEMA
				GlobalVar.ModWrite.Qset := REAL_TO_INT(SPCModbus1.OutputQ*0.001);//JEMA
			{ELSE}	
				Hugo4 := 2;
				GlobalVar.ModWrite.OutWset := SPCModbus1.OutputP; //ABG
				GlobalVar.ModWrite.OutVArSet := SPCModbus1.OutputQ;	//ABG
			{END_IF}
		
		ELSE
		//Reset functions
			{IF defined (JEMA)}
				Hugo5 := 1;
				GlobalVar.ModWrite.Pset :=0; //JEMA
				GlobalVar.ModWrite.Qset := 0;	//JEMA
			{ELSE}	
				Hugo5 := 2;
				GlobalVar.ModWrite.OutWset := 0; //JEMA
				GlobalVar.ModWrite.OutVArSet := 0;	//JEMA
			{END_IF}
			
		END_IF
	//Heart Beat send to DSP through Modbus
		GlobalVar.ModWrite.HeartBeat := INT_TO_UINT(GlobalVar.wMiliseconds);
		PreviousHeartBeat := GlobalVar.ModRead.HeartBeat;
	//Miliseconds tick for determining the scan cycle
		Tp := Globalvar.wMiliseconds;	
	//Write Modbus Registers
		mWritecounter := 0;
		{IF defined (JEMA)}
			Hugo6 := 1;
			ipAddr  := '192.168.1.51';
		{ELSE}	
			Hugo6 := 2;
			ipAddr  := '10.200.8.195';
		{END_IF}
		
		fbWriteRegs.sIPAddr :=ipAddr;
		fbWriteRegs.nQuantity := (*SIZEOF(Communications.ModWriteNRG)/2;*) SIZEOF(GlobalVar.ModWrite)/2; 
		{IF defined (JEMA)}
			Hugo7 := 1;
			fbWriteRegs.nMBAddr :=  16#1AD;(*JEMA*)
			//fbReadRegs.nMBAddr :=*16#0000;*)(*NRGLab*)
			//fbReadRegs.nMBAddr := 16#8064;//ABENGOA Memory location read
		{ELSE}	
			Hugo7 := 2;
			fbWriteRegs.nMBAddr := 16#4000; //LUA-FEC 
		{END_IF}
	
		fbWriteRegs.cbLength := (*SIZEOF(Communications.ModWriteNRG);*) SIZEOF(GlobalVar.ModWrite);
		fbWriteRegs.pSrcAddr := (*ADR(Communications.ModWriteNRG);*) ADR(GlobalVar.ModWrite);
		fbWriteRegs.tTimeout := T#5S;
		fbWriteRegs(bExecute:=TRUE);
	ELSE 
		fbWriteRegs(bExecute:=FALSE);
		IF fbwriteregs.bBusy THEN
		mWritecounter := mWritecounter + 1;
		END_IF
		
	END_IF
//End of Write Modbus Slave

	IF GlobalVar.ModRead.HeartBeat = FECHeartBeat THEN
		CounterCommFailure := CounterCommFailure + 1;
			IF CounterCommFailure > 10 THEN
				GlobalVar.CommunicationFailureModbus := TRUE;
				CounterCommFailure := 0;
			END_IF
	ELSE
		GlobalVar.CommunicationFailureModbus := FALSE;
		CounterCommFailure := 0;
	END_IF
	
	FECHeartBeat := GlobalVar.ModRead.HeartBeat;

////////////////////////////////////////////Event recorder
eventcnt := eventcnt + 1;
IF eventcnt = 2 THEN
	eventcnt := 0;

	EventRecorder_in_modbus.BatSoc := Globalvar.ModRead.BatSoc;
	{IF defined (JEMA)}
		Hugo8 := 1;
		EventRecorder_in_modbus.Vdc := GlobalVar.ModRead.CtrlPriority;
	{ELSE}	
		Hugo8 := 2;
		EventRecorder_in_modbus.Vdc := Globalvar.ModRead.SM_ManualControl;
	{END_IF}

	EventRecorder_in_modbus.TotW := Globalvar.ModRead.TotW;
	EventRecorder_in_modbus.TotVar := Globalvar.ModRead.TotVar;
	EventRecorder_in_modbus.GridFre := Globalvar.ModRead.GridFre;
	EventRecorder_in_modbus.Vrms := Globalvar.ModRead.Vrmsa;
	EventRecorder_in_modbus.Irms := Globalvar.ModRead.Irmsa;
	
	gvl.fbHistorian.ListeningRecording_IN_Modbus(HistorianDataPacket := EventRecorder_in_modbus);
	
	IF  communications.EtherCAT_Inputs.Command < 4 THEN
		EventRecorderControlOut.Pout_Inertia := Communications.PowerOfService.InertiaEmulationP_Service;
		EventRecorderControlOut.Pout_FrequencyRegulation := Communications.PowerOfService.FrequencyRegulationP_Service;
		EventRecorderControlOut.Pout_ModelFrequencyAttenuation := Communications.PowerOfService.ModalFreqAttP_Service;
		EventRecorderControlOut.Qout_VoltageRegulation := Communications.PowerOfService.VoltageRegulationQ_Service;
		EventRecorderControlOut.Pref := SPCModbus1.OutputP;
		EventRecorderControlOut.Qref := SPCModbus1.OutputQ;	
	
		gvl.fbHistorian.ListeningRecording_ControlOut(HistorianDataPacket := EventRecorderControlOut);
	END_IF
END_IF

END_PROGRAM

// ---- Functions/ModReadScaling.TcPOU
FUNCTION ModReadScaling : int
VAR_INPUT
END_VAR
VAR
END_VAR

GlobalVar.ScaledModRead.GridFre := INT_TO_REAL(GlobalVar.ModRead.GridFre)*0.01;

GlobalVar.ScaledModRead.Irmsa := INT_TO_REAL(GlobalVar.ModRead.Irmsa)*0.1;
GlobalVar.ScaledModRead.Irmsb := INT_TO_REAL(GlobalVar.ModRead.Irmsb)*0.1;
GlobalVar.ScaledModRead.Irmsc := INT_TO_REAL(GlobalVar.ModRead.Irmsc)*0.1;

GlobalVar.ScaledModRead.Vrmsa := INT_TO_REAL(GlobalVar.ModRead.Vrmsa)*0.1;
GlobalVar.ScaledModRead.Vrmsb := INT_TO_REAL(GlobalVar.ModRead.Vrmsb)*0.1;
GlobalVar.ScaledModRead.Vrmsc := INT_TO_REAL(GlobalVar.ModRead.Vrmsc)*0.1;
//GlobalVar.ScaledModRead.Vdc := INT_TO_REAL(GlobalVar.ModRead.Vdc)*0.1;
//GlobalVar.ScaledModRead.Idc := INT_TO_REAL(GlobalVar.ModRead.Idc)*0.1;

GlobalVar.ScaledModRead.TotW := INT_TO_REAL(GlobalVar.ModRead.TotW)*100.0;
GlobalVar.ScaledModRead.TotVar := INT_TO_REAL(GlobalVar.ModRead.TotVar)*100.0;

//GlobalVar.ScaledModRead.Vd := INT_TO_REAL(GlobalVar.ModRead.Vd)*0.1;
//GlobalVar.ScaledModRead.Vq := INT_TO_REAL(GlobalVar.ModRead.Vq)*0.1;

//GlobalVar.ScaledModRead.fbOpMode := GlobalVar.ModRead.fbOpMode;
//GlobalVar.ScaledModRead.OpMode := GlobalVar.ModRead.OpMode;

GlobalVar.ScaledModRead.GrAlm0 := GlobalVar.ModRead.GrAlm0;
GlobalVar.ScaledModRead.GrAlm1 := GlobalVar.ModRead.GrAlm1;
GlobalVar.ScaledModRead.GrAlm2 := GlobalVar.ModRead.GrAlm2;
GlobalVar.ScaledModRead.GrAlm3 := GlobalVar.ModRead.GrAlm3;
GlobalVar.ScaledModRead.GrAlm4 := GlobalVar.ModRead.GrAlm4;

END_FUNCTION

// ---- Functions/Communications/EtherCAT_MappingModbus.TcPOU
FUNCTION EtherCAT_MappingModbus : bool
VAR_INPUT
	Modbus_Controller : POINTER TO modbus_SPC;
	
END_VAR
VAR
END_VAR

//Commands
	//Common Block - Commands
		Modbus_Controller^.ActivePowerLimitation := Communications.EtherCAT_Commands.CommonBlock.Bits.ActivePowerLimitation;
		Modbus_Controller^.ReactivePowerLimitation := Communications.EtherCAT_Commands.CommonBlock.Bits.ReactivePowerLimitation;
		Modbus_Controller^.State_Of_Health := Communications.EtherCAT_Commands.CommonBlock.Bits.State_Of_Health;
		Modbus_Controller^.Reset_To_Default_Common := Communications.EtherCAT_Commands.CommonBlock.Bits.Reset_To_Default_Common; //Check how to do this
		
	//Inertia Emulation - Commands
		Modbus_Controller^.Enable_Inertia := Communications.EtherCAT_Commands.InertiaEmulation.Bits.Enable_Inertia;
		Modbus_Controller^.Inertia_Reset_States := Communications.EtherCAT_Commands.InertiaEmulation.Bits.Inertia_Reset_States;
		Modbus_Controller^.Limit_ROCOF := Communications.EtherCAT_Commands.InertiaEmulation.Bits.Limit_ROCOF;
		Modbus_Controller^.Delta_Power_Limit_Inertia := Communications.EtherCAT_Commands.InertiaEmulation.Bits.Delta_Power_Limit_Inertia;
		Modbus_Controller^.Reset_To_Default_Inertia := Communications.EtherCAT_Commands.InertiaEmulation.Bits.Reset_To_Default_Inertia; //Chechk how to do this
	
	//Frequency Regulation - Commands
		Modbus_Controller^.Enable_DroopP := Communications.EtherCAT_Commands.FrequencyRegulation.Bits.Enable_DroopP;
		Modbus_Controller^.Delta_Power_Limit_FreqRegulation := Communications.EtherCAT_Commands.FrequencyRegulation.Bits.Delta_Power_Limit_FreqRegulation;
		Modbus_Controller^.DeadBandLimitationP := Communications.EtherCAT_Commands.FrequencyRegulation.Bits.DeadBandLimitationP;
		Modbus_Controller^.Delta_Energy_Limit := Communications.EtherCAT_Commands.FrequencyRegulation.Bits.Delta_Energy_Limit;
		Modbus_Controller^.Reset_Energy_State := Communications.EtherCAT_Commands.FrequencyRegulation.Bits.Reset_Energy_State;
		Modbus_Controller^.Reset_To_Default_FreqRegulation := Communications.EtherCAT_Commands.FrequencyRegulation.Bits.Reset_To_Default_FreqRegulation; //Check How to do this.
		
	//Modal Frequency Attenuation - Commands
		Modbus_Controller^.Enable_ModalFreq := Communications.EtherCAT_Commands.ModalFreq.Bits.Enable_ModalFreq;
		Modbus_Controller^.Delta_Power_Limit_modalFreq := Communications.EtherCAT_Commands.ModalFreq.Bits.Delta_Power_Limit_ModalFreq;
		Modbus_Controller^.DeadBandLimitationV := Communications.EtherCAT_Commands.VoltageRegulation.Bits.DeadBandLimitationV;
		Modbus_Controller^.Reset_To_Default_ModalFreq := Communications.EtherCAT_Commands.ModalFreq.Bits.Reset_To_Default_ModalFreq;//Check How to do this.
	
	//Voltage Regulation - Commands
		Modbus_Controller^.Enable_VoltageRef := Communications.EtherCAT_Commands.VoltageRegulation.Bits.Enable_VoltageRef;
		Modbus_Controller^.Delta_Power_Limit_Voltage := Communications.EtherCAT_Commands.VoltageRegulation.Bits.Delta_Power_Limit_Voltage;
		Modbus_Controller^.Reset_To_Default_VoltageReg := Communications.EtherCAT_Commands.VoltageRegulation.Bits.Reset_To_Default_VoltageReg;//Check How to do this.
		
//parameters
	//Common Block - Parameters
		Modbus_Controller^.NominalPower := Communications.EhterCAT_Parameters.CommonBlock_Params.NominalPower;
		Modbus_Controller^.NominalFreq := Communications.EhterCAT_Parameters.CommonBlock_Params.NominalFreq;
		Modbus_Controller^.NominalVoltage := Communications.EhterCAT_Parameters.CommonBlock_Params.NominalVoltage;
		Modbus_Controller^.ActivePowerLimit := Communications.EhterCAT_Parameters.CommonBlock_Params.ActivePowerLimit;
		Modbus_Controller^.ReactivePowerLimit := Communications.EhterCAT_Parameters.CommonBlock_Params.ReactivePowerLimit;
		
	//Inertia Emulation - Parameters
		Modbus_Controller^.Inertia_Constant := Communications.EhterCAT_Parameters.InertiaEmulation_Params.Inertia_Constant;
		Modbus_Controller^.HighPassFilterConst := Communications.EhterCAT_Parameters.InertiaEmulation_Params.HighPassFilterConst;
		Modbus_Controller^.Max_ROCOF := Communications.EhterCAT_Parameters.InertiaEmulation_Params.Max_ROCOF;
		Modbus_Controller^.PowerLimit_Inertia := Communications.EhterCAT_Parameters.InertiaEmulation_Params.PowerLimit_Inertia;
		
	//frequency Regulation - Parameters
		Modbus_Controller^.DroopConstantP := Communications.EhterCAT_Parameters.FrequencyRegulation_Params.DroopConstantP;
		Modbus_Controller^.Max_Delta_Energy := Communications.EhterCAT_Parameters.FrequencyRegulation_Params.Max_delta_Energy;
		Modbus_Controller^.PowerLimit_Freq := Communications.EhterCAT_Parameters.FrequencyRegulation_Params.PowerLimit_Freq;
		Modbus_Controller^.FrequencyCutOff := Communications.EhterCAT_Parameters.FrequencyRegulation_Params.FrequencyCutOff;
		Modbus_Controller^.FreqDeadBand := Communications.EhterCAT_Parameters.FrequencyRegulation_Params.FreqDeadBand;
		
	//Modal Frequency Attenuation - Parameters
		Modbus_Controller^.ModalFreq_Gain := Communications.EhterCAT_Parameters.ModalFrequency_Params.ModalFreq_Gain;
		Modbus_Controller^.BandPassFilter_CenterFreq := Communications.EhterCAT_Parameters.ModalFrequency_Params.BandPassFilter_CenterFreq;
		Modbus_Controller^.PowerLimit_ModalFreq := Communications.EhterCAT_Parameters.ModalFrequency_Params.PowerLimit_ModalFreq;
		Modbus_Controller^.VoltageCutOff := Communications.EhterCAT_Parameters.VoltageRegulation_Params.VoltageCutOff;
		Modbus_Controller^.VoltDeadBand := Communications.EhterCAT_Parameters.VoltageRegulation_Params.VoltDeadBand;
		
	//Voltage Regulation
		Modbus_Controller^.DroopConstantV := Communications.EhterCAT_Parameters.VoltageRegulation_Params.DroopConstantV;
		Modbus_Controller^.PowerLimit_Voltage := Communications.EhterCAT_Parameters.VoltageRegulation_Params.PowerLimit_Voltage;

END_FUNCTION

// ---- Programs/State_Machine.TcPOU
PROGRAM State_Machine
VAR
	//Data Send 2 FEC
		DataSend2FEC 		AT %Q*		: data_16real;
		
	//Data Received
		DataReceived AT %I*: data_16real;

	//Current state of FLC
		CurrentState : eCurrentState;

		// Current State of FEC
		FEC_CurrState : eFEC_CurrState;
		
		P_mod_ref : REAL;
		Q_mod_ref : REAL;
		
		RampDown : REAL := 1;
	wAutoManCtl: INT;
	
	Hugo :REAL;
	Hugo1 : INT;
	Hugo2 : INT;
	Hugo3: INT;
	Hugo4: INT;
	
			
	EtherCATHeartBeat : DINT;
	CounterCommFailure : INT;
	
	
	TIMER_TIMEOUT:TON;	// Timer for enabling TLC communication
	TS_TIMEOUT: TIME;
	Counter_TimeOUT : INT;
	TS_WARNING: TIME;
	EmergencyStop_TimeOut	:	BOOL;
	Counter_TimeOUT_2	:	INT;
END_VAR

// Protection for EtherCAT
	IF Communications.EtherCAT_Inputs_DINT.Heartbeat = EtherCATHeartBeat THEN
		CounterCommFailure := CounterCommFailure + 1;
			IF CounterCommFailure > 500 THEN
				Communications.EtherCAT_Inputs_DINT.Command := 0;
				GlobalVar.CommunicationFailureEtherCAT := TRUE;
				Communications.EtherCAT_Variables.WarningLog.Bits.EtherCAT_Failure := TRUE;
				CounterCommFailure := 0;
			END_IF
	ELSE
		GlobalVar.CommunicationFailureEtherCAT := FALSE;
		Communications.EtherCAT_Variables.WarningLog.Bits.EtherCAT_Failure := FALSE;
		CounterCommFailure := 0;
	END_IF
	EtherCATHeartBeat := Communications.EtherCAT_Inputs_DINT.Heartbeat;
// End of protection for EtherCAT


{IF defined (JEMA)}
	Hugo1 := 1;
	Mapping_ModbusReadRegisters(ADR(GlobalVar.ScaledModRead),ADR(Communications.EtherCAT_Monitor_Variables),ADR(Communications.EtherCAT_Variables));	
	Mapping_ModbusWriteRegisters(ADR(GlobalVar.ModWrite),ADR(Communications.EtherCAT_Inputs));
{ELSE}	
	Hugo1 := 2;
	GlobalVar.ModWrite.wAutoManCtl := REAL_TO_UINT(Communications.EtherCAT_Inputs.Command);
{END_IF}

//Rempaing from DINT To REAL and from REAL TO DINT.
Remap_EtherCAT_Variables(ADR(Communications.EhterCAT_Parameters_DINT),
						ADR(Communications.EtherCAT_EAP_Parameters_DINT),
						ADR(Communications.EtherCAT_Inputs_DINT),
						ADR(Communications.EtherCAT_Monitor_Variables_DINT),
						ADR(Communications.EhterCAT_Parameters),
						ADR(Communications.EtherCAT_EAP_Parameters),
						ADR(Communications.EtherCAT_Inputs),
						ADR(Communications.EtherCAT_Monitor_Variables));
			
//Read state machine of the Front End Controller.
		{IF defined (JEMA)}
			Hugo2 := 1;
			//Read state machine OF the Front End Controller.
			IF GlobalVar.ModRead.CtrlPriority = 1 THEN
				FEC_CurrState := UINT_TO_INT(GlobalVar.ModRead.fbOpMode);
			ELSE
				FEC_CurrState := 2;
			END_IF
		{ELSE}	
			Hugo2 := 2;
			FEC_CurrState := UINT_TO_INT(GlobalVar.ModRead.DerOpMode);
		{END_IF}
		
	IF GlobalVar.CommunicationFailureModbus = 1 THEN
		FEC_CurrState := 0;
	END_IF
					
//ALARMS FROM THE POWER CONVERTER.		

{IF defined (JEMA)}
	Hugo3 := 3;
	IF GlobalVar.ModRead.GrAlm0 > 0 THEN
		FEC_CurrState := 0;				
	END_IF
	IF GlobalVar.ModRead.GrAlm1 > 0 THEN
		FEC_CurrState := 0;				
	END_IF
	IF GlobalVar.ModRead.GrAlm2 > 0 THEN
		FEC_CurrState := 0;				
	END_IF
	IF GlobalVar.ModRead.GrAlm3 > 0 THEN
		FEC_CurrState := 0;				
	END_IF
	IF GlobalVar.ModRead.GrAlm4 > 0 THEN
		FEC_CurrState := 0;				
	END_IF
{ELSE}	
	Hugo3 := 2;
{END_IF}

//State Machine - First Level Controller
	CASE FEC_CurrState OF
		eFEC_CurrState.FEC_OFF:
			CurrentState := eCurrentState.OFF;
			GlobalVar.ModbusSPC_Enable := FALSE;
			GlobalVar.EAP_SPC_Enable := FALSE;
			
		eFEC_CurrState.FEC_STANDBY:
			CurrentState := eCurrentState.STANDBY;
			GlobalVar.ModbusSPC_Enable := FALSE;
			GlobalVar.EAP_SPC_Enable := FALSE;
			
		eFEC_CurrState.FEC_MANUAL:
			CurrentState := eCurrentState.STANDBY;
			GlobalVar.ModbusSPC_Enable := FALSE;
			GlobalVar.EAP_SPC_Enable := FALSE;
			
		eFEC_CurrState.FEC_AVG_PWR_CTR:
			CurrentState := eCurrentState.AVG_PWR_CTR;
			GlobalVar.ModbusSPC_Enable := TRUE;
			GlobalVar.EAP_SPC_Enable := FALSE;
			
		eFEC_CurrState.FEC_INST_PWR_CTR:
			CurrentState := eCurrentState.INST_PWR_CTR;
			GlobalVar.ModbusSPC_Enable := FALSE;
			
			IF GlobalVar.CommunicationFailureEtherCAT = FALSE THEN
				GlobalVar.EAP_SPC_Enable := TRUE;
			ELSE
				GlobalVar.EAP_SPC_Enable := FALSE;
			END_IF
	ELSE
		CurrentState := eCurrentState.STANDBY;	
	END_CASE
	
	{IF defined (JEMA)}
		Hugo := 1;
		Mapping_Monitoring_Variables(GlobalVar.ScaledModRead,ADR(Communications.EtherCAT_Monitor_Variables),ADR(Communications.EtherCAT_Variables));
	{ELSE}
		Hugo := 2;
		Mapping_Monitoring_Variables_ABG(GlobalVar.ModRead,ADR(Communications.EtherCAT_Monitor_Variables),ADR(Communications.EtherCAT_Variables));
	{END_IF}
	

//////////Alarms/Warnings of our system
	TS_TIMEOUT := STRING_TO_TIME(INSERT('T#ms','1000',2));
	TIMER_TIMEOUT(IN:= NOT TIMER_TIMEOUT.Q, PT:= TS_TIMEOUT);
	
	IF GlobalVar.CommunicationFailureModbus = TRUE THEN
		Communications.EtherCAT_Variables.WarningLog.Bits.ModbusComm_FLC_PCS := TRUE;	
	ELSE
		Communications.EtherCAT_Variables.WarningLog.Bits.ModbusComm_FLC_PCS := FALSE;	
	END_IF
	

	IF (Communications.EtherCAT_Inputs.Command <> Communications.EtherCAT_Variables.Status) AND  Communications.EtherCAT_Inputs.Command <> 100 THEN
		IF TIMER_TIMEOUT.Q THEN
			Counter_TimeOUT := Counter_TimeOUT + 1;
		END_IF
		IF Counter_TimeOUT = 120 THEN
			Communications.EtherCAT_Variables.WarningLog.Bits.CommandTimeout := TRUE; 
			Counter_TimeOUT := 0;
		END_IF
	ELSE 
		IF TIMER_TIMEOUT.Q THEN
			Counter_TimeOUT_2 := Counter_TimeOUT_2 + 1;
		END_IF
		
		IF Counter_TimeOUT_2 = 300 THEN
			Communications.EtherCAT_Variables.WarningLog.Bits.CommandTimeout := FALSE; 
			Counter_TimeOUT_2 := 0;
		END_IF	
		Counter_TimeOUT := 0;
	END_IF
	
	IF Communications.EtherCAT_Monitor_Variables.Vrmsa > Communications.EhterCAT_Parameters.CommonBlock_Params.NominalVoltage*1.4 THEN
		Communications.EtherCAT_Variables.WarningLog.Bits.OverVoltage := TRUE;
	ELSE
		Communications.EtherCAT_Variables.WarningLog.Bits.OverVoltage := FALSE;
	END_IF
	
	IF Communications.EtherCAT_Monitor_Variables.Vrmsa < Communications.EhterCAT_Parameters.CommonBlock_Params.NominalVoltage*0.5 THEN
		Communications.EtherCAT_Variables.WarningLog.Bits.UnderVoltage := TRUE;
	ELSE
		Communications.EtherCAT_Variables.WarningLog.Bits.UnderVoltage := FALSE;
	END_IF
	
	IF Communications.EtherCAT_Monitor_Variables.Irmsa > Communications.EhterCAT_Parameters.CommonBlock_Params.NominalPower/(3*(Communications.EhterCAT_Parameters.CommonBlock_Params.NominalVoltage+1)) THEN
		Communications.EtherCAT_Variables.WarningLog.Bits.OverCurrent := TRUE;
	ELSE
		Communications.EtherCAT_Variables.WarningLog.Bits.OverCurrent := FALSE;
	END_IF
	
	IF Communications.EtherCAT_Monitor_Variables.GridFre*0.1591549430918 > (Communications.EhterCAT_Parameters.CommonBlock_Params.NominalFreq +  Communications.EhterCAT_Parameters.CommonBlock_Params.NominalFreq*0.02) THEN
		Communications.EtherCAT_Variables.WarningLog.Bits.OverFrequency := TRUE;
	ELSE
		Communications.EtherCAT_Variables.WarningLog.Bits.OverFrequency := FALSE;
	END_IF
	
	IF Communications.EtherCAT_Monitor_Variables.GridFre*0.1591549430918 < (Communications.EhterCAT_Parameters.CommonBlock_Params.NominalFreq - Communications.EhterCAT_Parameters.CommonBlock_Params.NominalFreq*0.02) THEN
		Communications.EtherCAT_Variables.WarningLog.Bits.UnderFrequency := TRUE;
	ELSE
		Communications.EtherCAT_Variables.WarningLog.Bits.UnderFrequency := FALSE;
	END_IF
	
	IF Communications.PowerOfService.InertiaEmulationP_Service > Communications.EhterCAT_Parameters.InertiaEmulation_Params.PowerLimit_Inertia THEN
		Communications.EtherCAT_Variables.WarningLog.Bits.Inertia_Overrange := TRUE;
	ELSE
		Communications.EtherCAT_Variables.WarningLog.Bits.Inertia_Overrange := FALSE;
	END_IF 
	
	IF Communications.PowerOfService.FrequencyRegulationP_Service > Communications.EhterCAT_Parameters.FrequencyRegulation_Params.PowerLimit_Freq THEN
		Communications.EtherCAT_Variables.WarningLog.Bits.Frequency_Overrange := TRUE;
	ELSE
		Communications.EtherCAT_Variables.WarningLog.Bits.Frequency_Overrange := FALSE;
	END_IF
	
	IF Communications.PowerOfService.VoltageRegulationQ_Service > Communications.EhterCAT_Parameters.VoltageRegulation_Params.PowerLimit_Voltage THEN
		Communications.EtherCAT_Variables.WarningLog.Bits.VoltReg_Overrange := TRUE;
	ELSE
		Communications.EtherCAT_Variables.WarningLog.Bits.VoltReg_Overrange := FALSE;
	END_IF
	
	IF Communications.PowerOfService.ModalFreqAttP_Service > Communications.EhterCAT_Parameters.ModalFrequency_Params.PowerLimit_ModalFreq THEN
		Communications.EtherCAT_Variables.WarningLog.Bits.ModFreq_Overrange := TRUE;
	ELSE
		Communications.EtherCAT_Variables.WarningLog.Bits.ModFreq_Overrange := FALSE;
	END_IF
	
	IF Communications.EtherCAT_Monitor_Variables.BatSoc > 80 THEN
		Communications.EtherCAT_Variables.WarningLog.Bits.Battery_80Perc := TRUE;
	ELSE
		Communications.EtherCAT_Variables.WarningLog.Bits.Battery_80Perc := FALSE;
	END_IF
	
	IF Communications.EtherCAT_Monitor_Variables.BatSoc < 20 THEN
		Communications.EtherCAT_Variables.WarningLog.Bits.Battery_20Perc := TRUE;
	ELSE
		Communications.EtherCAT_Variables.WarningLog.Bits.Battery_20Perc := FALSE;
	END_IF
	
	
	/////////////////////Critical warnings
	IF Communications.EtherCAT_Variables.WarningLog.Bits.ModbusComm_FLC_PCS = TRUE THEN
		Communications.EtherCAT_Inputs.Command := 0;
		Communications.EtherCAT_Variables.Status := 0;
	END_IF
	
	IF Communications.EtherCAT_Variables.WarningLog.Bits.CommandTimeout = TRUE THEN
		Communications.EtherCAT_Inputs.Command := 0;
	END_IF
	
	IF Communications.EtherCAT_Variables.WarningLog.Bits.EtherCAT_Failure = TRUE THEN
		Communications.EtherCAT_Inputs.Command := 0;
		Communications.EtherCAT_Variables.Status := 0;
	END_IF

END_PROGRAM

// ---- Functions/Mapping_ModbusReadRegisters.TcPOU
FUNCTION Mapping_ModbusReadRegisters
VAR_INPUT
	Read_Struct : POINTER TO ScaledModRead;
	ToSLCVariables : POINTER TO EtherCAT_Monitor_Variables;
	ToSLCStatus : POINTER TO EtherCAT_Stat_Variables;
	
END_VAR
VAR
END_VAR

//Variables
	//Status Parameter
		ToSLCStatus^.Status := Read_Struct^.fbOpMode;				// This data block is for send modbus FLC-SLC
	//Battery parameters
		ToSLCVariables^.BatSoc := Read_Struct^.BatSoc;
		//ToSLCVariables^.BatSocUpLim := Read_Struct^.BatSocUpLimit;
		//ToSLCVariables^.BatSocLowLim := Read_Struct^.BatSocLowLimit;
	//Active and Reactive Power Reference
		ToSLCVariables^.TotW := Read_Struct^.TotW;
		ToSLCVariables^.TotVAr := Read_Struct^.TotVAr;
	//Grid Frequency
		ToSLCVariables^.GridFre := Read_Struct^.GridFre;
	//Grid Currents RMS
		ToSLCVariables^.Irmsa := Read_Struct^.Irmsa;
		ToSLCVariables^.Irmsb := Read_Struct^.Irmsb;
		ToSLCVariables^.Irmsc := Read_Struct^.Irmsc;
	//Grid Voltages RMS
		ToSLCVariables^.Vrmsa := Read_Struct^.Vrmsa;
		ToSLCVariables^.Vrmsb := Read_Struct^.Vrmsb;
		ToSLCVariables^.Vrmsc := Read_Struct^.Vrmsc;
	//HeartBeat reading
		ToSLCStatus^.HeartBeat := Read_Struct^.HeartBeat;

END_FUNCTION

// ---- Functions/Mapping_ModbusWriteRegisters.TcPOU
FUNCTION Mapping_ModbusWriteRegisters : bool
VAR_INPUT
	//Modbus_Structure : POINTER TO MOdbusWrite_NRG;
	Modbus_Structure : POINTER TO ModbusWrite;
	FromSLC : POINTER TO EtherCAT_Inputs;
END_VAR
VAR
	wAutoManCtl: INT;
END_VAR

//Commands
	//State machine operation
		Modbus_Structure^.CmdOpMode := REAL_TO_INT(FromSLC^.Command);
	//Power Reference
		//Modbus_Structure^.Pset := (FromSLC^.ActivePowerReference);
		//Modbus_Structure^.Qset := (FromSLC^.ReactivePowerReference);

//GlobalVar.ModWrite.SLC_Debugger := FromSLC^.Commands;

END_FUNCTION

// ---- Functions/Communications/Remap_EtherCAT_Variables.TcPOU
FUNCTION Remap_EtherCAT_Variables : BOOL
VAR_INPUT
	//Inputs
	Modbus_para_DINT 	: POINTER TO Parameters_DINT;
	EAP_para_DINT 		: POINTER TO Parameters_EAP_DINT;
	EtherCAT_input_DINT	:	POINTER TO EtherCAT_Inputs_DINT;
	EtherCAT_monitor_DINT	:	POINTER TO EtherCAT_Monitor_Variables_DINT;
	
	//Outputs
	Modbus_paras 	: POINTER TO Parameters;
	EAP_paras 		: POINTER TO Parameters_EAP;
	EtherCAT_inputs	:	POINTER TO EtherCAT_Inputs;
	EtherCAT_monitor_var	:	POINTER TO EtherCAT_Monitor_Variables;
	
END_VAR
VAR
END_VAR

//Modbus Parameters
// Aditonal services
Modbus_paras^.AdditionalService_Params.Reserved1 := DINT_TO_REAL(Modbus_para_DINT^.AdditionalService_Params.Reserved1);
Modbus_paras^.AdditionalService_Params.Reserved2 := DINT_TO_REAL(Modbus_para_DINT^.AdditionalService_Params.Reserved2);
Modbus_paras^.AdditionalService_Params.Reserved3 := DINT_TO_REAL(Modbus_para_DINT^.AdditionalService_Params.Reserved3);
Modbus_paras^.AdditionalService_Params.Reserved4 := DINT_TO_REAL(Modbus_para_DINT^.AdditionalService_Params.Reserved4);
Modbus_paras^.AdditionalService_Params.Reserved5 := DINT_TO_REAL(Modbus_para_DINT^.AdditionalService_Params.Reserved5);
Modbus_paras^.AdditionalService_Params.Reserved6 := DINT_TO_REAL(Modbus_para_DINT^.AdditionalService_Params.Reserved6);
Modbus_paras^.AdditionalService_Params.Reserved7 := DINT_TO_REAL(Modbus_para_DINT^.AdditionalService_Params.Reserved7);
Modbus_paras^.AdditionalService_Params.Reserved8 := DINT_TO_REAL(Modbus_para_DINT^.AdditionalService_Params.Reserved8);
Modbus_paras^.AdditionalService_Params.Reserved9 := DINT_TO_REAL(Modbus_para_DINT^.AdditionalService_Params.Reserved9);
Modbus_paras^.AdditionalService_Params.Reserved10 := DINT_TO_REAL(Modbus_para_DINT^.AdditionalService_Params.Reserved10);
Modbus_paras^.AdditionalService_Params.Reserved11 := DINT_TO_REAL(Modbus_para_DINT^.AdditionalService_Params.Reserved11);
Modbus_paras^.AdditionalService_Params.Reserved12 := DINT_TO_REAL(Modbus_para_DINT^.AdditionalService_Params.Reserved12);
Modbus_paras^.AdditionalService_Params.Reserved13 := DINT_TO_REAL(Modbus_para_DINT^.AdditionalService_Params.Reserved13);
Modbus_paras^.AdditionalService_Params.Reserved14 := DINT_TO_REAL(Modbus_para_DINT^.AdditionalService_Params.Reserved14);
Modbus_paras^.AdditionalService_Params.Reserved15 := DINT_TO_REAL(Modbus_para_DINT^.AdditionalService_Params.Reserved15);
Modbus_paras^.AdditionalService_Params.Reserved16 := DINT_TO_REAL(Modbus_para_DINT^.AdditionalService_Params.Reserved16);
//CommonBlock_Params
Modbus_paras^.CommonBlock_Params.ActivePowerLimit := DINT_TO_REAL(Modbus_para_DINT^.CommonBlock_Params.ActivePowerLimit);
Modbus_paras^.CommonBlock_Params.NominalFreq := 0.01*DINT_TO_REAL(Modbus_para_DINT^.CommonBlock_Params.NominalFreq);
Modbus_paras^.CommonBlock_Params.NominalPower := DINT_TO_REAL(Modbus_para_DINT^.CommonBlock_Params.NominalPower);
Modbus_paras^.CommonBlock_Params.NominalVoltage := 0.01*DINT_TO_REAL(Modbus_para_DINT^.CommonBlock_Params.NominalVoltage);
Modbus_paras^.CommonBlock_Params.ReactivePowerLimit := DINT_TO_REAL(Modbus_para_DINT^.CommonBlock_Params.ReactivePowerLimit);
Modbus_paras^.CommonBlock_Params.Reserved1 := DINT_TO_REAL(Modbus_para_DINT^.CommonBlock_Params.Reserved1);
Modbus_paras^.CommonBlock_Params.Reserved2 := DINT_TO_REAL(Modbus_para_DINT^.CommonBlock_Params.Reserved2);
Modbus_paras^.CommonBlock_Params.Reserved3 := DINT_TO_REAL(Modbus_para_DINT^.CommonBlock_Params.Reserved3);
Modbus_paras^.CommonBlock_Params.Reserved4 := DINT_TO_REAL(Modbus_para_DINT^.CommonBlock_Params.Reserved4);
Modbus_paras^.CommonBlock_Params.Reserved5 := DINT_TO_REAL(Modbus_para_DINT^.CommonBlock_Params.Reserved5);
Modbus_paras^.CommonBlock_Params.Reserved6 := DINT_TO_REAL(Modbus_para_DINT^.CommonBlock_Params.Reserved6);
Modbus_paras^.CommonBlock_Params.Reserved7 := DINT_TO_REAL(Modbus_para_DINT^.CommonBlock_Params.Reserved7);
Modbus_paras^.CommonBlock_Params.Reserved8 := DINT_TO_REAL(Modbus_para_DINT^.CommonBlock_Params.Reserved8);
Modbus_paras^.CommonBlock_Params.Reserved9 := DINT_TO_REAL(Modbus_para_DINT^.CommonBlock_Params.Reserved9);
Modbus_paras^.CommonBlock_Params.Reserved10 := DINT_TO_REAL(Modbus_para_DINT^.CommonBlock_Params.Reserved10);
Modbus_paras^.CommonBlock_Params.Reserved11 := DINT_TO_REAL(Modbus_para_DINT^.CommonBlock_Params.Reserved11);
//FrequencyRegulation_Params
Modbus_paras^.FrequencyRegulation_Params.DroopConstantP := DINT_TO_REAL(Modbus_para_DINT^.FrequencyRegulation_Params.DroopConstantP)*0.1;
Modbus_paras^.FrequencyRegulation_Params.FreqDeadBand := DINT_TO_REAL(Modbus_para_DINT^.FrequencyRegulation_Params.FreqDeadBand)*0.1;
Modbus_paras^.FrequencyRegulation_Params.FrequencyCutOff := DINT_TO_REAL(Modbus_para_DINT^.FrequencyRegulation_Params.FrequencyCutOff)*0.01;
Modbus_paras^.FrequencyRegulation_Params.Max_delta_Energy := DINT_TO_REAL(Modbus_para_DINT^.FrequencyRegulation_Params.Max_delta_Energy);
Modbus_paras^.FrequencyRegulation_Params.PowerLimit_Freq := DINT_TO_REAL(Modbus_para_DINT^.FrequencyRegulation_Params.PowerLimit_Freq);
Modbus_paras^.FrequencyRegulation_Params.Reserved1 := DINT_TO_REAL(Modbus_para_DINT^.FrequencyRegulation_Params.Reserved1);
Modbus_paras^.FrequencyRegulation_Params.Reserved2 := DINT_TO_REAL(Modbus_para_DINT^.FrequencyRegulation_Params.Reserved2);
Modbus_paras^.FrequencyRegulation_Params.Reserved3 := DINT_TO_REAL(Modbus_para_DINT^.FrequencyRegulation_Params.Reserved3);
Modbus_paras^.FrequencyRegulation_Params.Reserved4 := DINT_TO_REAL(Modbus_para_DINT^.FrequencyRegulation_Params.Reserved4);
Modbus_paras^.FrequencyRegulation_Params.Reserved5 := DINT_TO_REAL(Modbus_para_DINT^.FrequencyRegulation_Params.Reserved5);
Modbus_paras^.FrequencyRegulation_Params.Reserved6 := DINT_TO_REAL(Modbus_para_DINT^.FrequencyRegulation_Params.Reserved6);
Modbus_paras^.FrequencyRegulation_Params.Reserved7 := DINT_TO_REAL(Modbus_para_DINT^.FrequencyRegulation_Params.Reserved7);
Modbus_paras^.FrequencyRegulation_Params.Reserved8 := DINT_TO_REAL(Modbus_para_DINT^.FrequencyRegulation_Params.Reserved8);
Modbus_paras^.FrequencyRegulation_Params.Reserved9 := DINT_TO_REAL(Modbus_para_DINT^.FrequencyRegulation_Params.Reserved9);
Modbus_paras^.FrequencyRegulation_Params.Reserved10 := DINT_TO_REAL(Modbus_para_DINT^.FrequencyRegulation_Params.Reserved10);
Modbus_paras^.FrequencyRegulation_Params.Reserved11 := DINT_TO_REAL(Modbus_para_DINT^.FrequencyRegulation_Params.Reserved11);

//InertiaEmulation_Params
Modbus_paras^.InertiaEmulation_Params.HighPassFilterConst := DINT_TO_REAL(Modbus_para_DINT^.InertiaEmulation_Params.HighPassFilterConst)*0.01;
Modbus_paras^.InertiaEmulation_Params.Inertia_Constant := DINT_TO_REAL(Modbus_para_DINT^.InertiaEmulation_Params.Inertia_Constant)*0.1;
Modbus_paras^.InertiaEmulation_Params.Max_ROCOF := DINT_TO_REAL(Modbus_para_DINT^.InertiaEmulation_Params.Max_ROCOF)*0.1;
Modbus_paras^.InertiaEmulation_Params.PowerLimit_Inertia := DINT_TO_REAL(Modbus_para_DINT^.InertiaEmulation_Params.PowerLimit_Inertia);
Modbus_paras^.InertiaEmulation_Params.Reserved1 := DINT_TO_REAL(Modbus_para_DINT^.InertiaEmulation_Params.Reserved1);
Modbus_paras^.InertiaEmulation_Params.Reserved2 := DINT_TO_REAL(Modbus_para_DINT^.InertiaEmulation_Params.Reserved2);
Modbus_paras^.InertiaEmulation_Params.Reserved3 := DINT_TO_REAL(Modbus_para_DINT^.InertiaEmulation_Params.Reserved3);
Modbus_paras^.InertiaEmulation_Params.Reserved4 := DINT_TO_REAL(Modbus_para_DINT^.InertiaEmulation_Params.Reserved4);
Modbus_paras^.InertiaEmulation_Params.Reserved5 := DINT_TO_REAL(Modbus_para_DINT^.InertiaEmulation_Params.Reserved5);
Modbus_paras^.InertiaEmulation_Params.Reserved6 := DINT_TO_REAL(Modbus_para_DINT^.InertiaEmulation_Params.Reserved6);
Modbus_paras^.InertiaEmulation_Params.Reserved7 := DINT_TO_REAL(Modbus_para_DINT^.InertiaEmulation_Params.Reserved7);
Modbus_paras^.InertiaEmulation_Params.Reserved8 := DINT_TO_REAL(Modbus_para_DINT^.InertiaEmulation_Params.Reserved8);
Modbus_paras^.InertiaEmulation_Params.Reserved9 := DINT_TO_REAL(Modbus_para_DINT^.InertiaEmulation_Params.Reserved9);
Modbus_paras^.InertiaEmulation_Params.Reserved10 := DINT_TO_REAL(Modbus_para_DINT^.InertiaEmulation_Params.Reserved10);
Modbus_paras^.InertiaEmulation_Params.Reserved11 := DINT_TO_REAL(Modbus_para_DINT^.InertiaEmulation_Params.Reserved11);
Modbus_paras^.InertiaEmulation_Params.Reserved12 := DINT_TO_REAL(Modbus_para_DINT^.InertiaEmulation_Params.Reserved12);

//InertiaEmulation_Params
Modbus_paras^.ModalFrequency_Params.BandPassFilter_CenterFreq := DINT_TO_REAL(Modbus_para_DINT^.ModalFrequency_Params.BandPassFilter_CenterFreq)*0.1;
Modbus_paras^.ModalFrequency_Params.ModalFreq_Gain := DINT_TO_REAL(Modbus_para_DINT^.ModalFrequency_Params.ModalFreq_Gain)*0.1;
Modbus_paras^.ModalFrequency_Params.PowerLimit_ModalFreq := DINT_TO_REAL(Modbus_para_DINT^.ModalFrequency_Params.PowerLimit_ModalFreq);
Modbus_paras^.ModalFrequency_Params.Reserved1 := DINT_TO_REAL(Modbus_para_DINT^.ModalFrequency_Params.Reserved1);
Modbus_paras^.ModalFrequency_Params.Reserved2 := DINT_TO_REAL(Modbus_para_DINT^.ModalFrequency_Params.Reserved2);
Modbus_paras^.ModalFrequency_Params.Reserved3 := DINT_TO_REAL(Modbus_para_DINT^.ModalFrequency_Params.Reserved3);
Modbus_paras^.ModalFrequency_Params.Reserved4 := DINT_TO_REAL(Modbus_para_DINT^.ModalFrequency_Params.Reserved4);
Modbus_paras^.ModalFrequency_Params.Reserved5 := DINT_TO_REAL(Modbus_para_DINT^.ModalFrequency_Params.Reserved5);
Modbus_paras^.ModalFrequency_Params.Reserved6 := DINT_TO_REAL(Modbus_para_DINT^.ModalFrequency_Params.Reserved6);
Modbus_paras^.ModalFrequency_Params.Reserved7 := DINT_TO_REAL(Modbus_para_DINT^.ModalFrequency_Params.Reserved7);
Modbus_paras^.ModalFrequency_Params.Reserved8 := DINT_TO_REAL(Modbus_para_DINT^.ModalFrequency_Params.Reserved8);
Modbus_paras^.ModalFrequency_Params.Reserved9 := DINT_TO_REAL(Modbus_para_DINT^.ModalFrequency_Params.Reserved9);
Modbus_paras^.ModalFrequency_Params.Reserved10 := DINT_TO_REAL(Modbus_para_DINT^.ModalFrequency_Params.Reserved10);
Modbus_paras^.ModalFrequency_Params.Reserved11 := DINT_TO_REAL(Modbus_para_DINT^.ModalFrequency_Params.Reserved11);
Modbus_paras^.ModalFrequency_Params.Reserved12 := DINT_TO_REAL(Modbus_para_DINT^.ModalFrequency_Params.Reserved12);
Modbus_paras^.ModalFrequency_Params.Reserved13 := DINT_TO_REAL(Modbus_para_DINT^.ModalFrequency_Params.Reserved13);

//VoltageRegulation_Params
Modbus_paras^.VoltageRegulation_Params.DroopConstantV := DINT_TO_REAL(Modbus_para_DINT^.VoltageRegulation_Params.DroopConstantV)*0.1;
Modbus_paras^.VoltageRegulation_Params.PowerLimit_Voltage := DINT_TO_REAL(Modbus_para_DINT^.VoltageRegulation_Params.PowerLimit_Voltage);
Modbus_paras^.VoltageRegulation_Params.VoltageCutOff := DINT_TO_REAL(Modbus_para_DINT^.VoltageRegulation_Params.VoltageCutOff)*0.01;
Modbus_paras^.VoltageRegulation_Params.VoltDeadBand := DINT_TO_REAL(Modbus_para_DINT^.VoltageRegulation_Params.VoltDeadBand)*0.1;
Modbus_paras^.VoltageRegulation_Params.Reserved1 := DINT_TO_REAL(Modbus_para_DINT^.VoltageRegulation_Params.Reserved1);
Modbus_paras^.VoltageRegulation_Params.Reserved2 := DINT_TO_REAL(Modbus_para_DINT^.VoltageRegulation_Params.Reserved2);
Modbus_paras^.VoltageRegulation_Params.Reserved3 := DINT_TO_REAL(Modbus_para_DINT^.VoltageRegulation_Params.Reserved3);
Modbus_paras^.VoltageRegulation_Params.Reserved4 := DINT_TO_REAL(Modbus_para_DINT^.VoltageRegulation_Params.Reserved4);
Modbus_paras^.VoltageRegulation_Params.Reserved5 := DINT_TO_REAL(Modbus_para_DINT^.VoltageRegulation_Params.Reserved5);
Modbus_paras^.VoltageRegulation_Params.Reserved6 := DINT_TO_REAL(Modbus_para_DINT^.VoltageRegulation_Params.Reserved6);
Modbus_paras^.VoltageRegulation_Params.Reserved7 := DINT_TO_REAL(Modbus_para_DINT^.VoltageRegulation_Params.Reserved7);
Modbus_paras^.VoltageRegulation_Params.Reserved8 := DINT_TO_REAL(Modbus_para_DINT^.VoltageRegulation_Params.Reserved8);
Modbus_paras^.VoltageRegulation_Params.Reserved9 := DINT_TO_REAL(Modbus_para_DINT^.VoltageRegulation_Params.Reserved9);
Modbus_paras^.VoltageRegulation_Params.Reserved10 := DINT_TO_REAL(Modbus_para_DINT^.VoltageRegulation_Params.Reserved10);
Modbus_paras^.VoltageRegulation_Params.Reserved11 := DINT_TO_REAL(Modbus_para_DINT^.VoltageRegulation_Params.Reserved11);
Modbus_paras^.VoltageRegulation_Params.Reserved12 := DINT_TO_REAL(Modbus_para_DINT^.VoltageRegulation_Params.Reserved12);

